LIN {X 0,Y 368.884,Z 241.032,A -85,B 0,C 180,E1 -12733.612,E2 -12733.612} C_VEL
LIN {X 0,Y 368.886,Z 241.019,A -85,B 0,C 180,E1 -12736.692,E2 -12736.692} C_VEL
LIN {X 0,Y 368.885,Z 241.034,A -85,B 0,C 180,E1 -12739.645,E2 -12739.645} C_VEL
LIN {X 0,Y 368.898,Z 241.029,A -85,B 0,C 180,E1 -12743.141,E2 -12743.141} C_VEL
LIN {X 0,Y 368.895,Z 241.032,A -85,B 0,C 180,E1 -12746.458,E2 -12746.458} C_VEL
LIN {X 0,Y 368.911,Z 241.032,A -85,B 0,C 180,E1 -12749.041,E2 -12749.041} C_VEL
LIN {X 0,Y 368.91,Z 241.028,A -85,B 0,C 180,E1 -12751.554,E2 -12751.554} C_VEL
LIN {X 0,Y 368.894,Z 241.03,A -85,B 0,C 180,E1 -12755.216,E2 -12755.216} C_VEL
LIN {X 0,Y 368.894,Z 241.03,A -85,B 0,C 180,E1 -12757.599,E2 -12757.599} C_VEL
LIN {X 0,Y 368.948,Z 241.029,A -85,B 0,C 180,E1 -12761.102,E2 -12761.102} C_VEL
LIN {X 0,Y 368.988,Z 241.017,A -85,B 0,C 180,E1 -12764.531,E2 -12764.531} C_VEL
LIN {X 0,Y 368.993,Z 241.012,A -85,B 0,C 180,E1 -12767.902,E2 -12767.902} C_VEL
LIN {X 0,Y 369.08,Z 241.007,A -85,B 0,C 180,E1 -12771.234,E2 -12771.234} C_VEL
LIN {X 0,Y 369.114,Z 241.004,A -85,B 0,C 180,E1 -12774.533,E2 -12774.533} C_VEL
LIN {X 0,Y 369.281,Z 240.983,A -85,B 0,C 180,E1 -12777.814,E2 -12777.814} C_VEL
LIN {X 0,Y 369.287,Z 240.982,A -85,B 0,C 180,E1 -12782.177,E2 -12782.177} C_VEL
LIN {X 0,Y 369.136,Z 241,A -85,B 0,C 180,E1 -12786.555,E2 -12786.555} C_VEL
LIN {X 0,Y 369.044,Z 241.011,A -85,B 0,C 180,E1 -12789.864,E2 -12789.864} C_VEL
LIN {X 0,Y 369.016,Z 241.014,A -85,B 0,C 180,E1 -12793.768,E2 -12793.768} C_VEL
LIN {X 0,Y 368.968,Z 241.023,A -85,B 0,C 180,E1 -12797.739,E2 -12797.739} C_VEL
LIN {X 0,Y 368.885,Z 241.034,A -85,B 0,C 180,E1 -12801.217,E2 -12801.217} C_VEL
LIN {X 0,Y 368.928,Z 241.026,A -85,B 0,C 180,E1 -12804.772,E2 -12804.772} C_VEL
LIN {X 0,Y 368.935,Z 241.026,A -85,B 0,C 180,E1 -12807.2,E2 -12807.2} C_VEL
LIN {X 0,Y 368.9,Z 241.033,A -85,B 0,C 180,E1 -12810.95,E2 -12810.95} C_VEL
LIN {X 0,Y 368.898,Z 241.029,A -85,B 0,C 180,E1 -12814.998,E2 -12814.998} C_VEL
LIN {X 0,Y 368.88,Z 241.032,A -85,B 0,C 180,E1 -12818.638,E2 -12818.638} C_VEL
LIN {X 0,Y 368.983,Z 241.215,A -85,B 0,C 180,E1 -12821.709,E2 -12821.709} C_VEL
LIN {X 0,Y 371.362,Z 251.966,A -85,B 0,C 180,E1 -12824.763,E2 -12824.763} C_VEL
LIN {X 0,Y 372.623,Z 259.108,A -85,B 0,C 180,E1 -12826.62,E2 -12826.62} C_VEL
LIN {X 0,Y 373.619,Z 263.254,A -85,B 0,C 180,E1 -12826.843,E2 -12826.843} C_VEL
LIN {X 0,Y 377.88,Z 282.484,A -85,B 0,C 180,E1 -12827.564,E2 -12827.564} C_VEL
LIN {X 0,Y 378.656,Z 288.482,A -85,B 0,C 180,E1 -12827.743,E2 -12827.743} C_VEL
LIN {X 0,Y 377.067,Z 367.322,A -85,B 0,C 180,E1 -12829.314,E2 -12829.314} C_VEL
LIN {X 0,Y 376.455,Z 380.341,A -85,B 0,C 180,E1 -12829.785,E2 -12829.785} C_VEL
LIN {X 0,Y 375.568,Z 393.469,A -85,B 0,C 180,E1 -12830.49,E2 -12830.49} C_VEL
LIN {X 0,Y 374.533,Z 405.678,A -85,B 0,C 180,E1 -12831.399,E2 -12831.399} C_VEL
LIN {X 0,Y 373.417,Z 416.7,A -85,B 0,C 180,E1 -12832.453,E2 -12832.453} C_VEL
LIN {X 0,Y 372.202,Z 426.94,A -85,B 0,C 180,E1 -12833.673,E2 -12833.673} C_VEL
LIN {X 0,Y 371.111,Z 436.307,A -85,B 0,C 180,E1 -12835.071,E2 -12835.071} C_VEL
LIN {X 0,Y 370.052,Z 444.979,A -85,B 0,C 180,E1 -12836.672,E2 -12836.672} C_VEL
LIN {X 0,Y 369.106,Z 452.589,A -85,B 0,C 180,E1 -12838.428,E2 -12838.428} C_VEL
LIN {X 0,Y 368.416,Z 458.773,A -85,B 0,C 180,E1 -12840.268,E2 -12840.268} C_VEL
LIN {X 0,Y 367.945,Z 463.489,A -85,B 0,C 180,E1 -12842.1,E2 -12842.1} C_VEL
LIN {X 0,Y 367.538,Z 466.997,A -85,B 0,C 180,E1 -12843.977,E2 -12843.977} C_VEL
LIN {X 0,Y 367.326,Z 468.508,A -85,B 0,C 180,E1 -12845.109,E2 -12845.109} C_VEL
LIN {X 0,Y 367.174,Z 469.903,A -85,B 0,C 180,E1 -12846.729,E2 -12846.729} C_VEL
LIN {X 0,Y 367.102,Z 470.42,A -85,B 0,C 180,E1 -12848.672,E2 -12848.672} C_VEL
LIN {X 0,Y 367.154,Z 470.118,A -85,B 0,C 180,E1 -12849.848,E2 -12849.848} C_VEL
LIN {X 0,Y 367.164,Z 469.396,A -85,B 0,C 180,E1 -12851.012,E2 -12851.012} C_VEL
LIN {X 0,Y 367.341,Z 467.033,A -85,B 0,C 180,E1 -12853.037,E2 -12853.037} C_VEL
LIN {X 0,Y 367.635,Z 463.214,A -85,B 0,C 180,E1 -12855.046,E2 -12855.046} C_VEL
LIN {X 0,Y 367.968,Z 458.316,A -85,B 0,C 180,E1 -12856.896,E2 -12856.896} C_VEL
LIN {X 0,Y 368.487,Z 451.945,A -85,B 0,C 180,E1 -12858.728,E2 -12858.728} C_VEL
LIN {X 0,Y 369.092,Z 444.484,A -85,B 0,C 180,E1 -12860.411,E2 -12860.411} C_VEL
LIN {X 0,Y 369.877,Z 436.445,A -85,B 0,C 180,E1 -12861.876,E2 -12861.876} C_VEL
LIN {X 0,Y 370.717,Z 426.62,A -85,B 0,C 180,E1 -12863.334,E2 -12863.334} C_VEL
LIN {X 0,Y 371.696,Z 416.058,A -85,B 0,C 180,E1 -12864.577,E2 -12864.577} C_VEL
LIN {X 0,Y 372.649,Z 404.329,A -85,B 0,C 180,E1 -12865.675,E2 -12865.675} C_VEL
LIN {X 0,Y 373.338,Z 393.146,A -85,B 0,C 180,E1 -12866.493,E2 -12866.493} C_VEL
LIN {X 0,Y 374.013,Z 380.48,A -85,B 0,C 180,E1 -12867.174,E2 -12867.174} C_VEL
LIN {X 0,Y 374.519,Z 367.44,A -85,B 0,C 180,E1 -12867.649,E2 -12867.649} C_VEL
LIN {X 0,Y 375.577,Z 299.972,A -85,B 0,C 180,E1 -12868.986,E2 -12868.986} C_VEL
LIN {X 0,Y 375.805,Z 285.428,A -85,B 0,C 180,E1 -12869.266,E2 -12869.266} C_VEL
LIN {X 0,Y 371.349,Z 259.539,A -85,B 0,C 180,E1 -12870.036,E2 -12870.036} C_VEL
LIN {X 0,Y 371.475,Z 257.113,A -85,B 0,C 180,E1 -12870.544,E2 -12870.544} C_VEL
LIN {X 0,Y 371.516,Z 253.896,A -85,B 0,C 180,E1 -12871.357,E2 -12871.357} C_VEL
LIN {X 0,Y 369.913,Z 245.755,A -85,B 0,C 180,E1 -12873.542,E2 -12873.542} C_VEL
LIN {X 0,Y 369.638,Z 244.48,A -85,B 0,C 180,E1 -12873.89,E2 -12873.89} C_VEL
LIN {X 0,Y 368.97,Z 242.94,A -85,B 0,C 180,E1 -12874.434,E2 -12874.434} C_VEL
LIN {X 0,Y 367.348,Z 241.756,A -85,B 0,C 180,E1 -12875.294,E2 -12875.294} C_VEL
LIN {X 0,Y 365.439,Z 241.465,A -85,B 0,C 180,E1 -12876.173,E2 -12876.173} C_VEL
LIN {X 0,Y 363.108,Z 241.757,A -85,B 0,C 180,E1 -12877.399,E2 -12877.399} C_VEL
LIN {X 0,Y 362.124,Z 241.878,A -85,B 0,C 180,E1 -12878.345,E2 -12878.345} C_VEL
LIN {X 0,Y 362.031,Z 241.885,A -85,B 0,C 180,E1 -12878.665,E2 -12878.665} C_VEL
LIN {X 0,Y 361.927,Z 241.898,A -85,B 0,C 180,E1 -12882.335,E2 -12882.335} C_VEL
LIN {X 0,Y 361.925,Z 241.898,A -85,B 0,C 180,E1 -12884.624,E2 -12884.624} C_VEL
LIN {X 0,Y 361.92,Z 241.902,A -85,B 0,C 180,E1 -12888.103,E2 -12888.103} C_VEL
LIN {X 0,Y 361.82,Z 241.915,A -85,B 0,C 180,E1 -12891.659,E2 -12891.659} C_VEL
LIN {X 0,Y 361.836,Z 241.909,A -85,B 0,C 180,E1 -12895.299,E2 -12895.299} C_VEL
LIN {X 0,Y 361.825,Z 241.91,A -85,B 0,C 180,E1 -12899.078,E2 -12899.078} C_VEL
LIN {X 0,Y 361.818,Z 241.912,A -85,B 0,C 180,E1 -12902.95,E2 -12902.95} C_VEL
LIN {X 0,Y 361.836,Z 241.909,A -85,B 0,C 180,E1 -12905.642,E2 -12905.642} C_VEL
LIN {X 0,Y 361.799,Z 241.915,A -85,B 0,C 180,E1 -12909.022,E2 -12909.022} C_VEL
LIN {X 0,Y 361.805,Z 241.917,A -85,B 0,C 180,E1 -12912.835,E2 -12912.835} C_VEL
LIN {X 0,Y 361.795,Z 241.914,A -85,B 0,C 180,E1 -12915.952,E2 -12915.952} C_VEL
LIN {X 0,Y 361.794,Z 241.917,A -85,B 0,C 180,E1 -12919.254,E2 -12919.254} C_VEL
LIN {X 0,Y 361.846,Z 241.914,A -85,B 0,C 180,E1 -12922.987,E2 -12922.987} C_VEL
LIN {X 0,Y 361.844,Z 241.91,A -85,B 0,C 180,E1 -12926.637,E2 -12926.637} C_VEL
LIN {X 0,Y 361.836,Z 241.911,A -85,B 0,C 180,E1 -12929.675,E2 -12929.675} C_VEL
LIN {X 0,Y 361.846,Z 241.913,A -85,B 0,C 180,E1 -12933.473,E2 -12933.473} C_VEL
LIN {X 0,Y 361.868,Z 241.909,A -85,B 0,C 180,E1 -12937.149,E2 -12937.149} C_VEL
LIN {X 0,Y 361.88,Z 241.904,A -85,B 0,C 180,E1 -12940.727,E2 -12940.727} C_VEL
LIN {X 0,Y 361.941,Z 241.897,A -85,B 0,C 180,E1 -12944.231,E2 -12944.231} C_VEL
LIN {X 0,Y 361.999,Z 241.889,A -85,B 0,C 180,E1 -12946.533,E2 -12946.533} C_VEL
LIN {X 0,Y 361.997,Z 241.895,A -85,B 0,C 180,E1 -12949.942,E2 -12949.942} C_VEL
LIN {X 0,Y 362.122,Z 241.874,A -85,B 0,C 180,E1 -12953.318,E2 -12953.318} C_VEL
LIN {X 0,Y 362.27,Z 241.858,A -85,B 0,C 180,E1 -12957.781,E2 -12957.781} C_VEL
LIN {X 0,Y 362.207,Z 241.863,A -85,B 0,C 180,E1 -12961.116,E2 -12961.116} C_VEL
LIN {X 0,Y 362.265,Z 241.863,A -85,B 0,C 180,E1 -12962.228,E2 -12962.228} C_VEL
LIN {X 0,Y 362.128,Z 241.876,A -85,B 0,C 180,E1 -12966.691,E2 -12966.691} C_VEL
LIN {X 0,Y 362.008,Z 241.89,A -85,B 0,C 180,E1 -12970.067,E2 -12970.067} C_VEL
LIN {X 0,Y 362.011,Z 241.888,A -85,B 0,C 180,E1 -12973.902,E2 -12973.902} C_VEL
LIN {X 0,Y 361.942,Z 241.9,A -85,B 0,C 180,E1 -12976.937,E2 -12976.937} C_VEL
LIN {X 0,Y 361.901,Z 241.904,A -85,B 0,C 180,E1 -12980.464,E2 -12980.464} C_VEL
LIN {X 0,Y 361.909,Z 241.9,A -85,B 0,C 180,E1 -12984.115,E2 -12984.115} C_VEL
LIN {X 0,Y 361.851,Z 241.908,A -85,B 0,C 180,E1 -12987.787,E2 -12987.787} C_VEL
LIN {X 0,Y 361.864,Z 241.911,A -85,B 0,C 180,E1 -12991.287,E2 -12991.287} C_VEL
LIN {X 0,Y 361.87,Z 241.905,A -85,B 0,C 180,E1 -12994.282,E2 -12994.282} C_VEL
LIN {X 0,Y 361.876,Z 241.909,A -85,B 0,C 180,E1 -12997.223,E2 -12997.223} C_VEL
LIN {X 0,Y 361.827,Z 241.911,A -85,B 0,C 180,E1 -13000.752,E2 -13000.752} C_VEL
LIN {X 0,Y 361.827,Z 241.91,A -85,B 0,C 180,E1 -13004.371,E2 -13004.371} C_VEL
LIN {X 0,Y 361.839,Z 241.914,A -85,B 0,C 180,E1 -13007.572,E2 -13007.572} C_VEL
LIN {X 0,Y 361.86,Z 241.91,A -85,B 0,C 180,E1 -13011.572,E2 -13011.572} C_VEL
LIN {X 0,Y 361.891,Z 241.903,A -85,B 0,C 180,E1 -13014.656,E2 -13014.656} C_VEL
LIN {X 0,Y 361.855,Z 241.912,A -85,B 0,C 180,E1 -13018.371,E2 -13018.371} C_VEL
LIN {X 0,Y 361.932,Z 242.078,A -85,B 0,C 180,E1 -13021.906,E2 -13021.906} C_VEL
LIN {X 0,Y 363.903,Z 251.935,A -85,B 0,C 180,E1 -13024.549,E2 -13024.549} C_VEL
LIN {X 0,Y 364.929,Z 258.159,A -85,B 0,C 180,E1 -13026.143,E2 -13026.143} C_VEL
LIN {X 0,Y 364.18,Z 268.524,A -85,B 0,C 180,E1 -13028.594,E2 -13028.594} C_VEL
LIN {X 0,Y 364.736,Z 272.676,A -85,B 0,C 180,E1 -13028.775,E2 -13028.775} C_VEL
LIN {X 0,Y 368.963,Z 299.983,A -85,B 0,C 180,E1 -13029.539,E2 -13029.539} C_VEL
LIN {X 0,Y 367.671,Z 376.615,A -85,B 0,C 180,E1 -13031.072,E2 -13031.072} C_VEL
LIN {X 0,Y 367.097,Z 389.795,A -85,B 0,C 180,E1 -13031.548,E2 -13031.548} C_VEL
LIN {X 0,Y 366.391,Z 401.948,A -85,B 0,C 180,E1 -13032.198,E2 -13032.198} C_VEL
LIN {X 0,Y 365.439,Z 414.213,A -85,B 0,C 180,E1 -13033.088,E2 -13033.088} C_VEL
LIN {X 0,Y 364.526,Z 425.841,A -85,B 0,C 180,E1 -13034.196,E2 -13034.196} C_VEL
LIN {X 0,Y 363.631,Z 436.307,A -85,B 0,C 180,E1 -13035.447,E2 -13035.447} C_VEL
LIN {X 0,Y 362.755,Z 445.691,A -85,B 0,C 180,E1 -13036.84,E2 -13036.84} C_VEL
LIN {X 0,Y 361.837,Z 454.761,A -85,B 0,C 180,E1 -13038.515,E2 -13038.515} C_VEL
LIN {X 0,Y 361.209,Z 462.062,A -85,B 0,C 180,E1 -13040.196,E2 -13040.196} C_VEL
LIN {X 0,Y 360.825,Z 466.983,A -85,B 0,C 180,E1 -13041.598,E2 -13041.598} C_VEL
LIN {X 0,Y 360.511,Z 471.754,A -85,B 0,C 180,E1 -13043.281,E2 -13043.281} C_VEL
LIN {X 0,Y 360.358,Z 475.394,A -85,B 0,C 180,E1 -13044.963,E2 -13044.963} C_VEL
LIN {X 0,Y 360.28,Z 478.009,A -85,B 0,C 180,E1 -13046.643,E2 -13046.643} C_VEL
LIN {X 0,Y 360.23,Z 479.236,A -85,B 0,C 180,E1 -13047.762,E2 -13047.762} C_VEL
LIN {X 0,Y 360.256,Z 480.037,A -85,B 0,C 180,E1 -13048.88,E2 -13048.88} C_VEL
LIN {X 0,Y 360.281,Z 480.419,A -85,B 0,C 180,E1 -13049.998,E2 -13049.998} C_VEL
LIN {X 0,Y 360.254,Z 480.415,A -85,B 0,C 180,E1 -13051.116,E2 -13051.116} C_VEL
LIN {X 0,Y 360.229,Z 480.027,A -85,B 0,C 180,E1 -13052.234,E2 -13052.234} C_VEL
LIN {X 0,Y 360.283,Z 479.232,A -85,B 0,C 180,E1 -13053.353,E2 -13053.353} C_VEL
LIN {X 0,Y 360.385,Z 478.008,A -85,B 0,C 180,E1 -13054.472,E2 -13054.472} C_VEL
LIN {X 0,Y 360.463,Z 475.575,A -85,B 0,C 180,E1 -13056.072,E2 -13056.072} C_VEL
LIN {X 0,Y 360.789,Z 471.827,A -85,B 0,C 180,E1 -13057.835,E2 -13057.835} C_VEL
LIN {X 0,Y 361.299,Z 467.141,A -85,B 0,C 180,E1 -13059.515,E2 -13059.515} C_VEL
LIN {X 0,Y 362.125,Z 460.107,A -85,B 0,C 180,E1 -13061.472,E2 -13061.472} C_VEL
LIN {X 0,Y 363.127,Z 452.5,A -85,B 0,C 180,E1 -13063.143,E2 -13063.143} C_VEL
LIN {X 0,Y 364.392,Z 443.156,A -85,B 0,C 180,E1 -13064.772,E2 -13064.772} C_VEL
LIN {X 0,Y 365.496,Z 433.562,A -85,B 0,C 180,E1 -13066.13,E2 -13066.13} C_VEL
LIN {X 0,Y 366.714,Z 423.502,A -85,B 0,C 180,E1 -13067.279,E2 -13067.279} C_VEL
LIN {X 0,Y 367.828,Z 413.132,A -85,B 0,C 180,E1 -13068.23,E2 -13068.23} C_VEL
LIN {X 0,Y 368.965,Z 400.702,A -85,B 0,C 180,E1 -13069.108,E2 -13069.108} C_VEL
LIN {X 0,Y 369.847,Z 387.695,A -85,B 0,C 180,E1 -13069.782,E2 -13069.782} C_VEL
LIN {X 0,Y 370.553,Z 374.988,A -85,B 0,C 180,E1 -13070.207,E2 -13070.207} C_VEL
LIN {X 0,Y 371.946,Z 299.95,A -85,B 0,C 180,E1 -13071.731,E2 -13071.731} C_VEL
LIN {X 0,Y 368.448,Z 280.867,A -85,B 0,C 180,E1 -13072.405,E2 -13072.405} C_VEL
LIN {X 0,Y 365.677,Z 268.304,A -85,B 0,C 180,E1 -13072.932,E2 -13072.932} C_VEL
LIN {X 0,Y 366.148,Z 262.196,A -85,B 0,C 180,E1 -13074.371,E2 -13074.371} C_VEL
LIN {X 0,Y 364.501,Z 253.179,A -85,B 0,C 180,E1 -13076.829,E2 -13076.829} C_VEL
LIN {X 0,Y 361.897,Z 242.036,A -85,B 0,C 180,E1 -13080.093,E2 -13080.093} C_VEL
LIN {X 0,Y 361.859,Z 241.909,A -85,B 0,C 180,E1 -13084.277,E2 -13084.277} C_VEL
LIN {X 0,Y 361.864,Z 241.909,A -85,B 0,C 180,E1 -13087.219,E2 -13087.219} C_VEL
LIN {X 0,Y 361.833,Z 241.91,A -85,B 0,C 180,E1 -13090.751,E2 -13090.751} C_VEL
LIN {X 0,Y 361.818,Z 241.917,A -85,B 0,C 180,E1 -13094.365,E2 -13094.365} C_VEL
LIN {X 0,Y 361.831,Z 241.902,A -85,B 0,C 180,E1 -13097.566,E2 -13097.566} C_VEL
LIN {X 0,Y 361.843,Z 241.909,A -85,B 0,C 180,E1 -13101.568,E2 -13101.568} C_VEL
LIN {X 0,Y 361.873,Z 241.907,A -85,B 0,C 180,E1 -13104.652,E2 -13104.652} C_VEL
LIN {X 0,Y 361.836,Z 241.911,A -85,B 0,C 180,E1 -13108.367,E2 -13108.367} C_VEL
LIN {X 0,Y 361.863,Z 241.905,A -85,B 0,C 180,E1 -13110.948,E2 -13110.948} C_VEL
LIN {X 0,Y 361.863,Z 241.904,A -85,B 0,C 180,E1 -13114.701,E2 -13114.701} C_VEL
LIN {X 0,Y 361.849,Z 241.907,A -85,B 0,C 180,E1 -13118.341,E2 -13118.341} C_VEL
LIN {X 0,Y 361.914,Z 241.899,A -85,B 0,C 180,E1 -13122.081,E2 -13122.081} C_VEL
LIN {X 0,Y 361.954,Z 241.9,A -85,B 0,C 180,E1 -13125.375,E2 -13125.375} C_VEL
LIN {X 0,Y 361.958,Z 241.891,A -85,B 0,C 180,E1 -13128.8,E2 -13128.8} C_VEL
LIN {X 0,Y 362.075,Z 241.872,A -85,B 0,C 180,E1 -13132.187,E2 -13132.187} C_VEL
LIN {X 0,Y 362.087,Z 241.879,A -85,B 0,C 180,E1 -13134.427,E2 -13134.427} C_VEL
LIN {X 0,Y 362.243,Z 241.859,A -85,B 0,C 180,E1 -13137.772,E2 -13137.772} C_VEL
LIN {X 0,Y 362.25,Z 241.859,A -85,B 0,C 180,E1 -13142.219,E2 -13142.219} C_VEL
LIN {X 0,Y 362.1,Z 241.876,A -85,B 0,C 180,E1 -13146.683,E2 -13146.683} C_VEL
LIN {X 0,Y 361.98,Z 241.891,A -85,B 0,C 180,E1 -13150.059,E2 -13150.059} C_VEL
LIN {X 0,Y 361.977,Z 241.892,A -85,B 0,C 180,E1 -13153.894,E2 -13153.894} C_VEL
LIN {X 0,Y 361.905,Z 241.899,A -85,B 0,C 180,E1 -13156.93,E2 -13156.93} C_VEL
LIN {X 0,Y 361.862,Z 241.91,A -85,B 0,C 180,E1 -13160.457,E2 -13160.457} C_VEL
LIN {X 0,Y 361.867,Z 241.912,A -85,B 0,C 180,E1 -13164.109,E2 -13164.109} C_VEL
LIN {X 0,Y 361.914,Z 241.903,A -85,B 0,C 180,E1 -13166.717,E2 -13166.717} C_VEL
LIN {X 0,Y 361.843,Z 241.911,A -85,B 0,C 180,E1 -13170.324,E2 -13170.324} C_VEL
LIN {X 0,Y 361.823,Z 241.917,A -85,B 0,C 180,E1 -13174.277,E2 -13174.277} C_VEL
LIN {X 0,Y 361.84,Z 241.914,A -85,B 0,C 180,E1 -13177.221,E2 -13177.221} C_VEL
LIN {X 0,Y 361.925,Z 242.054,A -85,B 0,C 180,E1 -13181.221,E2 -13181.221} C_VEL
LIN {X 0,Y 364.082,Z 251.548,A -85,B 0,C 180,E1 -13184.013,E2 -13184.013} C_VEL
LIN {X 0,Y 365.584,Z 259.305,A -85,B 0,C 180,E1 -13186.095,E2 -13186.095} C_VEL
LIN {X 0,Y 367.171,Z 264.374,A -85,B 0,C 180,E1 -13186.373,E2 -13186.373} C_VEL
LIN {X 0,Y 371.549,Z 284.065,A -85,B 0,C 180,E1 -13187.135,E2 -13187.135} C_VEL
LIN {X 0,Y 372.244,Z 288.032,A -85,B 0,C 180,E1 -13187.272,E2 -13187.272} C_VEL
LIN {X 0,Y 370.567,Z 367.095,A -85,B 0,C 180,E1 -13188.876,E2 -13188.876} C_VEL
LIN {X 0,Y 369.964,Z 379.833,A -85,B 0,C 180,E1 -13189.339,E2 -13189.339} C_VEL
LIN {X 0,Y 369.075,Z 392.402,A -85,B 0,C 180,E1 -13190.011,E2 -13190.011} C_VEL
LIN {X 0,Y 368.166,Z 403.08,A -85,B 0,C 180,E1 -13190.78,E2 -13190.78} C_VEL
LIN {X 0,Y 366.943,Z 414.608,A -85,B 0,C 180,E1 -13191.844,E2 -13191.844} C_VEL
LIN {X 0,Y 365.696,Z 425.274,A -85,B 0,C 180,E1 -13193.092,E2 -13193.092} C_VEL
LIN {X 0,Y 364.511,Z 434.505,A -85,B 0,C 180,E1 -13194.427,E2 -13194.427} C_VEL
LIN {X 0,Y 363.477,Z 442.768,A -85,B 0,C 180,E1 -13195.896,E2 -13195.896} C_VEL
LIN {X 0,Y 362.533,Z 449.914,A -85,B 0,C 180,E1 -13197.458,E2 -13197.458} C_VEL
LIN {X 0,Y 361.725,Z 456.172,A -85,B 0,C 180,E1 -13199.158,E2 -13199.158} C_VEL
LIN {X 0,Y 361.097,Z 461.808,A -85,B 0,C 180,E1 -13201.13,E2 -13201.13} C_VEL
LIN {X 0,Y 360.696,Z 465.301,A -85,B 0,C 180,E1 -13202.751,E2 -13202.751} C_VEL
LIN {X 0,Y 360.309,Z 468.147,A -85,B 0,C 180,E1 -13204.59,E2 -13204.59} C_VEL
LIN {X 0,Y 360.078,Z 469.937,A -85,B 0,C 180,E1 -13206.525,E2 -13206.525} C_VEL
LIN {X 0,Y 360.017,Z 470.506,A -85,B 0,C 180,E1 -13208.231,E2 -13208.231} C_VEL
LIN {X 0,Y 360.047,Z 470.337,A -85,B 0,C 180,E1 -13209.526,E2 -13209.526} C_VEL
LIN {X 0,Y 360.049,Z 469.76,A -85,B 0,C 180,E1 -13210.622,E2 -13210.622} C_VEL
LIN {X 0,Y 360.09,Z 468.721,A -85,B 0,C 180,E1 -13211.805,E2 -13211.805} C_VEL
LIN {X 0,Y 360.231,Z 467.239,A -85,B 0,C 180,E1 -13212.986,E2 -13212.986} C_VEL
LIN {X 0,Y 360.477,Z 464.114,A -85,B 0,C 180,E1 -13214.742,E2 -13214.742} C_VEL
LIN {X 0,Y 360.873,Z 458.918,A -85,B 0,C 180,E1 -13216.814,E2 -13216.814} C_VEL
LIN {X 0,Y 361.406,Z 452.311,A -85,B 0,C 180,E1 -13218.789,E2 -13218.789} C_VEL
LIN {X 0,Y 362.029,Z 444.907,A -85,B 0,C 180,E1 -13220.504,E2 -13220.504} C_VEL
LIN {X 0,Y 362.939,Z 435.68,A -85,B 0,C 180,E1 -13222.211,E2 -13222.211} C_VEL
LIN {X 0,Y 363.795,Z 426.139,A -85,B 0,C 180,E1 -13223.624,E2 -13223.624} C_VEL
LIN {X 0,Y 364.839,Z 415.442,A -85,B 0,C 180,E1 -13224.89,E2 -13224.89} C_VEL
LIN {X 0,Y 365.827,Z 403.481,A -85,B 0,C 180,E1 -13226.014,E2 -13226.014} C_VEL
LIN {X 0,Y 366.604,Z 390.865,A -85,B 0,C 180,E1 -13226.911,E2 -13226.911} C_VEL
LIN {X 0,Y 367.296,Z 378.133,A -85,B 0,C 180,E1 -13227.569,E2 -13227.569} C_VEL
LIN {X 0,Y 367.743,Z 364.816,A -85,B 0,C 180,E1 -13228.017,E2 -13228.017} C_VEL
LIN {X 0,Y 369.04,Z 286.728,A -85,B 0,C 180,E1 -13229.566,E2 -13229.566} C_VEL
LIN {X 0,Y 364.472,Z 259.735,A -85,B 0,C 180,E1 -13230.382,E2 -13230.382} C_VEL
LIN {X 0,Y 364.479,Z 258.385,A -85,B 0,C 180,E1 -13230.609,E2 -13230.609} C_VEL
LIN {X 0,Y 364.573,Z 255.361,A -85,B 0,C 180,E1 -13231.382,E2 -13231.382} C_VEL
LIN {X 0,Y 362.982,Z 247.218,A -85,B 0,C 180,E1 -13233.609,E2 -13233.609} C_VEL
LIN {X 0,Y 362.022,Z 241.921,A -85,B 0,C 180,E1 -13235.153,E2 -13235.153} C_VEL
LIN {X 0,Y 362.076,Z 241.88,A -85,B 0,C 180,E1 -13238.186,E2 -13238.186} C_VEL
LIN {X 0,Y 362.031,Z 241.885,A -85,B 0,C 180,E1 -13238.665,E2 -13238.665} C_VEL
LIN {X 0,Y 361.311,Z 241.981,A -85,B 0,C 180,E1 -13239.593,E2 -13239.593} C_VEL
LIN {X 0,Y 358.39,Z 242.34,A -85,B 0,C 180,E1 -13241.1,E2 -13241.1} C_VEL
LIN {X 0,Y 355.965,Z 242.641,A -85,B 0,C 180,E1 -13242.32,E2 -13242.32} C_VEL
LIN {X 0,Y 354.964,Z 242.768,A -85,B 0,C 180,E1 -13243.265,E2 -13243.265} C_VEL
LIN {X 0,Y 354.902,Z 242.777,A -85,B 0,C 180,E1 -13243.584,E2 -13243.584} C_VEL
LIN {X 0,Y 354.862,Z 242.779,A -85,B 0,C 180,E1 -13247.284,E2 -13247.284} C_VEL
LIN {X 0,Y 354.791,Z 242.787,A -85,B 0,C 180,E1 -13250.891,E2 -13250.891} C_VEL
LIN {X 0,Y 354.78,Z 242.789,A -85,B 0,C 180,E1 -13254.584,E2 -13254.584} C_VEL
LIN {X 0,Y 354.77,Z 242.793,A -85,B 0,C 180,E1 -13258.39,E2 -13258.39} C_VEL
LIN {X 0,Y 354.755,Z 242.797,A -85,B 0,C 180,E1 -13262.338,E2 -13262.338} C_VEL
LIN {X 0,Y 354.79,Z 242.787,A -85,B 0,C 180,E1 -13265.703,E2 -13265.703} C_VEL
LIN {X 0,Y 354.744,Z 242.792,A -85,B 0,C 180,E1 -13269.417,E2 -13269.417} C_VEL
LIN {X 0,Y 354.758,Z 242.795,A -85,B 0,C 180,E1 -13272.871,E2 -13272.871} C_VEL
LIN {X 0,Y 354.744,Z 242.793,A -85,B 0,C 180,E1 -13276.108,E2 -13276.108} C_VEL
LIN {X 0,Y 354.747,Z 242.795,A -85,B 0,C 180,E1 -13279.181,E2 -13279.181} C_VEL
LIN {X 0,Y 354.783,Z 242.789,A -85,B 0,C 180,E1 -13282.41,E2 -13282.41} C_VEL
LIN {X 0,Y 354.794,Z 242.792,A -85,B 0,C 180,E1 -13284.946,E2 -13284.946} C_VEL
LIN {X 0,Y 354.778,Z 242.789,A -85,B 0,C 180,E1 -13288.412,E2 -13288.412} C_VEL
LIN {X 0,Y 354.779,Z 242.791,A -85,B 0,C 180,E1 -13291.619,E2 -13291.619} C_VEL
LIN {X 0,Y 354.797,Z 242.792,A -85,B 0,C 180,E1 -13295.425,E2 -13295.425} C_VEL
LIN {X 0,Y 354.821,Z 242.786,A -85,B 0,C 180,E1 -13299.118,E2 -13299.118} C_VEL
LIN {X 0,Y 354.878,Z 242.776,A -85,B 0,C 180,E1 -13302.724,E2 -13302.724} C_VEL
LIN {X 0,Y 354.951,Z 242.768,A -85,B 0,C 180,E1 -13306.26,E2 -13306.26} C_VEL
LIN {X 0,Y 354.953,Z 242.772,A -85,B 0,C 180,E1 -13309.74,E2 -13309.74} C_VEL
LIN {X 0,Y 355.088,Z 242.75,A -85,B 0,C 180,E1 -13313.185,E2 -13313.185} C_VEL
LIN {X 0,Y 355.232,Z 242.735,A -85,B 0,C 180,E1 -13317.737,E2 -13317.737} C_VEL
LIN {X 0,Y 355.176,Z 242.739,A -85,B 0,C 180,E1 -13321.138,E2 -13321.138} C_VEL
LIN {X 0,Y 355.227,Z 242.739,A -85,B 0,C 180,E1 -13322.272,E2 -13322.272} C_VEL
LIN {X 0,Y 355.095,Z 242.751,A -85,B 0,C 180,E1 -13326.824,E2 -13326.824} C_VEL
LIN {X 0,Y 354.965,Z 242.769,A -85,B 0,C 180,E1 -13330.269,E2 -13330.269} C_VEL
LIN {X 0,Y 354.956,Z 242.767,A -85,B 0,C 180,E1 -13334.022,E2 -13334.022} C_VEL
LIN {X 0,Y 354.904,Z 242.773,A -85,B 0,C 180,E1 -13338.095,E2 -13338.095} C_VEL
LIN {X 0,Y 354.829,Z 242.782,A -85,B 0,C 180,E1 -13342.11,E2 -13342.11} C_VEL
LIN {X 0,Y 354.864,Z 242.78,A -85,B 0,C 180,E1 -13344.58,E2 -13344.58} C_VEL
LIN {X 0,Y 354.813,Z 242.784,A -85,B 0,C 180,E1 -13348.388,E2 -13348.388} C_VEL
LIN {X 0,Y 354.803,Z 242.785,A -85,B 0,C 180,E1 -13352.336,E2 -13352.336} C_VEL
LIN {X 0,Y 354.838,Z 242.783,A -85,B 0,C 180,E1 -13355.701,E2 -13355.701} C_VEL
LIN {X 0,Y 354.786,Z 242.794,A -85,B 0,C 180,E1 -13359.414,E2 -13359.414} C_VEL
LIN {X 0,Y 354.798,Z 242.786,A -85,B 0,C 180,E1 -13362.867,E2 -13362.867} C_VEL
LIN {X 0,Y 354.778,Z 242.79,A -85,B 0,C 180,E1 -13366.103,E2 -13366.103} C_VEL
LIN {X 0,Y 354.779,Z 242.789,A -85,B 0,C 180,E1 -13369.176,E2 -13369.176} C_VEL
LIN {X 0,Y 354.817,Z 242.785,A -85,B 0,C 180,E1 -13372.405,E2 -13372.405} C_VEL
LIN {X 0,Y 354.829,Z 242.782,A -85,B 0,C 180,E1 -13374.941,E2 -13374.941} C_VEL
LIN {X 0,Y 354.81,Z 242.789,A -85,B 0,C 180,E1 -13378.405,E2 -13378.405} C_VEL
LIN {X 0,Y 354.889,Z 242.923,A -85,B 0,C 180,E1 -13381.621,E2 -13381.621} C_VEL
LIN {X 0,Y 356.836,Z 252.758,A -85,B 0,C 180,E1 -13384.321,E2 -13384.321} C_VEL
LIN {X 0,Y 357.922,Z 258.976,A -85,B 0,C 180,E1 -13385.954,E2 -13385.954} C_VEL
LIN {X 0,Y 357.45,Z 265.998,A -85,B 0,C 180,E1 -13387.68,E2 -13387.68} C_VEL
LIN {X 0,Y 357.318,Z 268.816,A -85,B 0,C 180,E1 -13388.274,E2 -13388.274} C_VEL
LIN {X 0,Y 359.225,Z 281.426,A -85,B 0,C 180,E1 -13388.678,E2 -13388.678} C_VEL
LIN {X 0,Y 362.172,Z 300.669,A -85,B 0,C 180,E1 -13389.226,E2 -13389.226} C_VEL
LIN {X 0,Y 360.856,Z 376.741,A -85,B 0,C 180,E1 -13390.774,E2 -13390.774} C_VEL
LIN {X 0,Y 360.26,Z 389.844,A -85,B 0,C 180,E1 -13391.258,E2 -13391.258} C_VEL
LIN {X 0,Y 359.529,Z 401.958,A -85,B 0,C 180,E1 -13391.92,E2 -13391.92} C_VEL
LIN {X 0,Y 358.639,Z 413.39,A -85,B 0,C 180,E1 -13392.757,E2 -13392.757} C_VEL
LIN {X 0,Y 357.648,Z 425.153,A -85,B 0,C 180,E1 -13393.883,E2 -13393.883} C_VEL
LIN {X 0,Y 356.726,Z 435.722,A -85,B 0,C 180,E1 -13395.158,E2 -13395.158} C_VEL
LIN {X 0,Y 355.794,Z 445.22,A -85,B 0,C 180,E1 -13396.578,E2 -13396.578} C_VEL
LIN {X 0,Y 354.843,Z 454.355,A -85,B 0,C 180,E1 -13398.285,E2 -13398.285} C_VEL
LIN {X 0,Y 354.186,Z 461.711,A -85,B 0,C 180,E1 -13400,E2 -13400} C_VEL
LIN {X 0,Y 353.762,Z 466.679,A -85,B 0,C 180,E1 -13401.429,E2 -13401.429} C_VEL
LIN {X 0,Y 353.43,Z 471.495,A -85,B 0,C 180,E1 -13403.146,E2 -13403.146} C_VEL
LIN {X 0,Y 353.263,Z 475.176,A -85,B 0,C 180,E1 -13404.862,E2 -13404.862} C_VEL
LIN {X 0,Y 353.204,Z 477.829,A -85,B 0,C 180,E1 -13406.576,E2 -13406.576} C_VEL
LIN {X 0,Y 353.141,Z 479.075,A -85,B 0,C 180,E1 -13407.717,E2 -13407.717} C_VEL
LIN {X 0,Y 353.155,Z 479.911,A -85,B 0,C 180,E1 -13408.858,E2 -13408.858} C_VEL
LIN {X 0,Y 353.182,Z 480.311,A -85,B 0,C 180,E1 -13409.998,E2 -13409.998} C_VEL
LIN {X 0,Y 353.154,Z 480.325,A -85,B 0,C 180,E1 -13411.139,E2 -13411.139} C_VEL
LIN {X 0,Y 353.208,Z 479.191,A -85,B 0,C 180,E1 -13413.42,E2 -13413.42} C_VEL
LIN {X 0,Y 353.3,Z 477.988,A -85,B 0,C 180,E1 -13414.562,E2 -13414.562} C_VEL
LIN {X 0,Y 353.363,Z 475.886,A -85,B 0,C 180,E1 -13416.021,E2 -13416.021} C_VEL
LIN {X 0,Y 353.74,Z 471.882,A -85,B 0,C 180,E1 -13417.992,E2 -13417.992} C_VEL
LIN {X 0,Y 354.281,Z 467.237,A -85,B 0,C 180,E1 -13419.706,E2 -13419.706} C_VEL
LIN {X 0,Y 355.149,Z 460.247,A -85,B 0,C 180,E1 -13421.701,E2 -13421.701} C_VEL
LIN {X 0,Y 356.228,Z 452.696,A -85,B 0,C 180,E1 -13423.402,E2 -13423.402} C_VEL
LIN {X 0,Y 357.519,Z 443.588,A -85,B 0,C 180,E1 -13425.041,E2 -13425.041} C_VEL
LIN {X 0,Y 358.701,Z 433.965,A -85,B 0,C 180,E1 -13426.444,E2 -13426.444} C_VEL
LIN {X 0,Y 359.979,Z 424.032,A -85,B 0,C 180,E1 -13427.613,E2 -13427.613} C_VEL
LIN {X 0,Y 361.138,Z 413.843,A -85,B 0,C 180,E1 -13428.58,E2 -13428.58} C_VEL
LIN {X 0,Y 362.325,Z 401.763,A -85,B 0,C 180,E1 -13429.472,E2 -13429.472} C_VEL
LIN {X 0,Y 363.221,Z 389.161,A -85,B 0,C 180,E1 -13430.159,E2 -13430.159} C_VEL
LIN {X 0,Y 364.037,Z 376.07,A -85,B 0,C 180,E1 -13430.628,E2 -13430.628} C_VEL
LIN {X 0,Y 365.518,Z 300.705,A -85,B 0,C 180,E1 -13432.194,E2 -13432.194} C_VEL
LIN {X 0,Y 361.522,Z 279.337,A -85,B 0,C 180,E1 -13432.978,E2 -13432.978} C_VEL
LIN {X 0,Y 358.999,Z 268.251,A -85,B 0,C 180,E1 -13433.467,E2 -13433.467} C_VEL
LIN {X 0,Y 359.27,Z 263.646,A -85,B 0,C 180,E1 -13434.561,E2 -13434.561} C_VEL
LIN {X 0,Y 357.309,Z 253.342,A -85,B 0,C 180,E1 -13437.445,E2 -13437.445} C_VEL
LIN {X 0,Y 354.879,Z 243.126,A -85,B 0,C 180,E1 -13440.493,E2 -13440.493} C_VEL
LIN {X 0,Y 354.805,Z 242.787,A -85,B 0,C 180,E1 -13440.996,E2 -13440.996} C_VEL
LIN {X 0,Y 354.812,Z 242.789,A -85,B 0,C 180,E1 -13443.699,E2 -13443.699} C_VEL
LIN {X 0,Y 354.801,Z 242.792,A -85,B 0,C 180,E1 -13446.457,E2 -13446.457} C_VEL
LIN {X 0,Y 354.803,Z 242.786,A -85,B 0,C 180,E1 -13449.415,E2 -13449.415} C_VEL
LIN {X 0,Y 354.788,Z 242.783,A -85,B 0,C 180,E1 -13452.863,E2 -13452.863} C_VEL
LIN {X 0,Y 354.767,Z 242.779,A -85,B 0,C 180,E1 -13456.1,E2 -13456.1} C_VEL
LIN {X 0,Y 354.767,Z 242.793,A -85,B 0,C 180,E1 -13459.172,E2 -13459.172} C_VEL
LIN {X 0,Y 354.8,Z 242.792,A -85,B 0,C 180,E1 -13462.401,E2 -13462.401} C_VEL
LIN {X 0,Y 354.811,Z 242.789,A -85,B 0,C 180,E1 -13464.937,E2 -13464.937} C_VEL
LIN {X 0,Y 354.792,Z 242.789,A -85,B 0,C 180,E1 -13468.401,E2 -13468.401} C_VEL
LIN {X 0,Y 354.797,Z 242.786,A -85,B 0,C 180,E1 -13471.611,E2 -13471.611} C_VEL
LIN {X 0,Y 354.802,Z 242.786,A -85,B 0,C 180,E1 -13475.416,E2 -13475.416} C_VEL
LIN {X 0,Y 354.82,Z 242.78,A -85,B 0,C 180,E1 -13479.109,E2 -13479.109} C_VEL
LIN {X 0,Y 354.873,Z 242.775,A -85,B 0,C 180,E1 -13482.715,E2 -13482.715} C_VEL
LIN {X 0,Y 354.943,Z 242.769,A -85,B 0,C 180,E1 -13486.251,E2 -13486.251} C_VEL
LIN {X 0,Y 354.944,Z 242.771,A -85,B 0,C 180,E1 -13489.731,E2 -13489.731} C_VEL
LIN {X 0,Y 355.092,Z 242.745,A -85,B 0,C 180,E1 -13493.176,E2 -13493.176} C_VEL
LIN {X 0,Y 355.205,Z 242.734,A -85,B 0,C 180,E1 -13497.728,E2 -13497.728} C_VEL
LIN {X 0,Y 355.129,Z 242.741,A -85,B 0,C 180,E1 -13501.13,E2 -13501.13} C_VEL
LIN {X 0,Y 355.212,Z 242.735,A -85,B 0,C 180,E1 -13502.263,E2 -13502.263} C_VEL
LIN {X 0,Y 355.067,Z 242.753,A -85,B 0,C 180,E1 -13506.816,E2 -13506.816} C_VEL
LIN {X 0,Y 354.936,Z 242.77,A -85,B 0,C 180,E1 -13510.26,E2 -13510.26} C_VEL
LIN {X 0,Y 354.922,Z 242.772,A -85,B 0,C 180,E1 -13514.014,E2 -13514.014} C_VEL
LIN {X 0,Y 354.867,Z 242.784,A -85,B 0,C 180,E1 -13518.088,E2 -13518.088} C_VEL
LIN {X 0,Y 354.794,Z 242.79,A -85,B 0,C 180,E1 -13521.414,E2 -13521.414} C_VEL
LIN {X 0,Y 354.834,Z 242.783,A -85,B 0,C 180,E1 -13524.572,E2 -13524.572} C_VEL
LIN {X 0,Y 354.854,Z 242.781,A -85,B 0,C 180,E1 -13527.092,E2 -13527.092} C_VEL
LIN {X 0,Y 354.77,Z 242.793,A -85,B 0,C 180,E1 -13530.995,E2 -13530.995} C_VEL
LIN {X 0,Y 354.776,Z 242.791,A -85,B 0,C 180,E1 -13533.698,E2 -13533.698} C_VEL
LIN {X 0,Y 354.769,Z 242.789,A -85,B 0,C 180,E1 -13536.456,E2 -13536.456} C_VEL
LIN {X 0,Y 354.872,Z 242.915,A -85,B 0,C 180,E1 -13540.708,E2 -13540.708} C_VEL
LIN {X 0,Y 357.04,Z 252.236,A -85,B 0,C 180,E1 -13543.538,E2 -13543.538} C_VEL
LIN {X 0,Y 358.457,Z 259.388,A -85,B 0,C 180,E1 -13545.52,E2 -13545.52} C_VEL
LIN {X 0,Y 360.825,Z 265.835,A -85,B 0,C 180,E1 -13545.9,E2 -13545.9} C_VEL
LIN {X 0,Y 365.19,Z 285.307,A -85,B 0,C 180,E1 -13546.68,E2 -13546.68} C_VEL
LIN {X 0,Y 365.824,Z 290.408,A -85,B 0,C 180,E1 -13546.841,E2 -13546.841} C_VEL
LIN {X 0,Y 364.084,Z 367.421,A -85,B 0,C 180,E1 -13548.432,E2 -13548.432} C_VEL
LIN {X 0,Y 363.413,Z 380.529,A -85,B 0,C 180,E1 -13548.921,E2 -13548.921} C_VEL
LIN {X 0,Y 362.52,Z 392.758,A -85,B 0,C 180,E1 -13549.594,E2 -13549.594} C_VEL
LIN {X 0,Y 361.483,Z 404.193,A -85,B 0,C 180,E1 -13550.443,E2 -13550.443} C_VEL
LIN {X 0,Y 360.196,Z 415.649,A -85,B 0,C 180,E1 -13551.545,E2 -13551.545} C_VEL
LIN {X 0,Y 358.813,Z 426.786,A -85,B 0,C 180,E1 -13552.902,E2 -13552.902} C_VEL
LIN {X 0,Y 357.6,Z 435.51,A -85,B 0,C 180,E1 -13554.222,E2 -13554.222} C_VEL
LIN {X 0,Y 356.38,Z 444.471,A -85,B 0,C 180,E1 -13555.909,E2 -13555.909} C_VEL
LIN {X 0,Y 355.311,Z 452.181,A -85,B 0,C 180,E1 -13557.722,E2 -13557.722} C_VEL
LIN {X 0,Y 354.489,Z 458.527,A -85,B 0,C 180,E1 -13559.634,E2 -13559.634} C_VEL
LIN {X 0,Y 353.917,Z 463.35,A -85,B 0,C 180,E1 -13561.54,E2 -13561.54} C_VEL
LIN {X 0,Y 353.46,Z 466.908,A -85,B 0,C 180,E1 -13563.463,E2 -13563.463} C_VEL
LIN {X 0,Y 353.099,Z 469.165,A -85,B 0,C 180,E1 -13565.295,E2 -13565.295} C_VEL
LIN {X 0,Y 353.004,Z 470.119,A -85,B 0,C 180,E1 -13566.538,E2 -13566.538} C_VEL
LIN {X 0,Y 352.916,Z 470.555,A -85,B 0,C 180,E1 -13567.77,E2 -13567.77} C_VEL
LIN {X 0,Y 352.938,Z 470.484,A -85,B 0,C 180,E1 -13569.356,E2 -13569.356} C_VEL
LIN {X 0,Y 352.962,Z 469.19,A -85,B 0,C 180,E1 -13571.425,E2 -13571.425} C_VEL
LIN {X 0,Y 353.114,Z 467.624,A -85,B 0,C 180,E1 -13572.79,E2 -13572.79} C_VEL
LIN {X 0,Y 353.352,Z 464.921,A -85,B 0,C 180,E1 -13574.426,E2 -13574.426} C_VEL
LIN {X 0,Y 353.657,Z 460.927,A -85,B 0,C 180,E1 -13576.206,E2 -13576.206} C_VEL
LIN {X 0,Y 354.051,Z 455.748,A -85,B 0,C 180,E1 -13577.972,E2 -13577.972} C_VEL
LIN {X 0,Y 354.622,Z 449.207,A -85,B 0,C 180,E1 -13579.727,E2 -13579.727} C_VEL
LIN {X 0,Y 355.45,Z 440.545,A -85,B 0,C 180,E1 -13581.559,E2 -13581.559} C_VEL
LIN {X 0,Y 356.281,Z 432.596,A -85,B 0,C 180,E1 -13582.92,E2 -13582.92} C_VEL
LIN {X 0,Y 357.248,Z 422.332,A -85,B 0,C 180,E1 -13584.357,E2 -13584.357} C_VEL
LIN {X 0,Y 358.363,Z 410.613,A -85,B 0,C 180,E1 -13585.644,E2 -13585.644} C_VEL
LIN {X 0,Y 359.262,Z 399.116,A -85,B 0,C 180,E1 -13586.637,E2 -13586.637} C_VEL
LIN {X 0,Y 360.003,Z 387.314,A -85,B 0,C 180,E1 -13587.414,E2 -13587.414} C_VEL
LIN {X 0,Y 360.626,Z 373.71,A -85,B 0,C 180,E1 -13588.047,E2 -13588.047} C_VEL
LIN {X 0,Y 360.988,Z 361.728,A -85,B 0,C 180,E1 -13588.398,E2 -13588.398} C_VEL
LIN {X 0,Y 362.234,Z 287.197,A -85,B 0,C 180,E1 -13589.896,E2 -13589.896} C_VEL
LIN {X 0,Y 357.562,Z 259.656,A -85,B 0,C 180,E1 -13590.748,E2 -13590.748} C_VEL
LIN {X 0,Y 357.625,Z 256.818,A -85,B 0,C 180,E1 -13591.409,E2 -13591.409} C_VEL
LIN {X 0,Y 356.044,Z 248.612,A -85,B 0,C 180,E1 -13593.68,E2 -13593.68} C_VEL
LIN {X 0,Y 355.045,Z 243.078,A -85,B 0,C 180,E1 -13595.255,E2 -13595.255} C_VEL
LIN {X 0,Y 355.049,Z 242.758,A -85,B 0,C 180,E1 -13595.682,E2 -13595.682} C_VEL
LIN {X 0,Y 354.992,Z 242.762,A -85,B 0,C 180,E1 -13598.65,E2 -13598.65} C_VEL
LIN {X 0,Y 354.887,Z 242.775,A -85,B 0,C 180,E1 -13602.584,E2 -13602.584} C_VEL
LIN {X 0,Y 354.902,Z 242.777,A -85,B 0,C 180,E1 -13603.584,E2 -13603.584} C_VEL
LIN {X 0,Y 354.291,Z 242.86,A -85,B 0,C 180,E1 -13604.531,E2 -13604.531} C_VEL
LIN {X 0,Y 351.463,Z 243.213,A -85,B 0,C 180,E1 -13606.07,E2 -13606.07} C_VEL
LIN {X 0,Y 349.014,Z 243.513,A -85,B 0,C 180,E1 -13607.315,E2 -13607.315} C_VEL
LIN {X 0,Y 347.932,Z 243.644,A -85,B 0,C 180,E1 -13608.279,E2 -13608.279} C_VEL
LIN {X 0,Y 347.829,Z 243.654,A -85,B 0,C 180,E1 -13608.606,E2 -13608.606} C_VEL
LIN {X 0,Y 347.716,Z 243.669,A -85,B 0,C 180,E1 -13612.585,E2 -13612.585} C_VEL
LIN {X 0,Y 347.713,Z 243.668,A -85,B 0,C 180,E1 -13615.118,E2 -13615.118} C_VEL
LIN {X 0,Y 347.706,Z 243.671,A -85,B 0,C 180,E1 -13617.705,E2 -13617.705} C_VEL
LIN {X 0,Y 347.705,Z 243.674,A -85,B 0,C 180,E1 -13620.354,E2 -13620.354} C_VEL
LIN {X 0,Y 347.72,Z 243.671,A -85,B 0,C 180,E1 -13624.048,E2 -13624.048} C_VEL
LIN {X 0,Y 347.728,Z 243.666,A -85,B 0,C 180,E1 -13627.327,E2 -13627.327} C_VEL
LIN {X 0,Y 347.671,Z 243.677,A -85,B 0,C 180,E1 -13630.307,E2 -13630.307} C_VEL
LIN {X 0,Y 347.698,Z 243.67,A -85,B 0,C 180,E1 -13633.414,E2 -13633.414} C_VEL
LIN {X 0,Y 347.704,Z 243.676,A -85,B 0,C 180,E1 -13636.692,E2 -13636.692} C_VEL
LIN {X 0,Y 347.684,Z 243.672,A -85,B 0,C 180,E1 -13640.188,E2 -13640.188} C_VEL
LIN {X 0,Y 347.739,Z 243.669,A -85,B 0,C 180,E1 -13642.684,E2 -13642.684} C_VEL
LIN {X 0,Y 347.735,Z 243.666,A -85,B 0,C 180,E1 -13645.962,E2 -13645.962} C_VEL
LIN {X 0,Y 347.724,Z 243.668,A -85,B 0,C 180,E1 -13649.656,E2 -13649.656} C_VEL
LIN {X 0,Y 347.726,Z 243.67,A -85,B 0,C 180,E1 -13653.605,E2 -13653.605} C_VEL
LIN {X 0,Y 347.745,Z 243.665,A -85,B 0,C 180,E1 -13656.165,E2 -13656.165} C_VEL
LIN {X 0,Y 347.782,Z 243.662,A -85,B 0,C 180,E1 -13659.913,E2 -13659.913} C_VEL
LIN {X 0,Y 347.83,Z 243.659,A -85,B 0,C 180,E1 -13663.574,E2 -13663.574} C_VEL
LIN {X 0,Y 347.888,Z 243.647,A -85,B 0,C 180,E1 -13667.166,E2 -13667.166} C_VEL
LIN {X 0,Y 347.936,Z 243.641,A -85,B 0,C 180,E1 -13670.706,E2 -13670.706} C_VEL
LIN {X 0,Y 348.04,Z 243.631,A -85,B 0,C 180,E1 -13674.21,E2 -13674.21} C_VEL
LIN {X 0,Y 348.194,Z 243.61,A -85,B 0,C 180,E1 -13677.691,E2 -13677.691} C_VEL
LIN {X 0,Y 348.145,Z 243.614,A -85,B 0,C 180,E1 -13681.161,E2 -13681.161} C_VEL
LIN {X 0,Y 348.188,Z 243.615,A -85,B 0,C 180,E1 -13682.318,E2 -13682.318} C_VEL
LIN {X 0,Y 348.062,Z 243.626,A -85,B 0,C 180,E1 -13686.963,E2 -13686.963} C_VEL
LIN {X 0,Y 347.905,Z 243.65,A -85,B 0,C 180,E1 -13690.479,E2 -13690.479} C_VEL
LIN {X 0,Y 347.913,Z 243.645,A -85,B 0,C 180,E1 -13694.153,E2 -13694.153} C_VEL
LIN {X 0,Y 347.844,Z 243.654,A -85,B 0,C 180,E1 -13698.262,E2 -13698.262} C_VEL
LIN {X 0,Y 347.782,Z 243.66,A -85,B 0,C 180,E1 -13701.629,E2 -13701.629} C_VEL
LIN {X 0,Y 347.782,Z 243.665,A -85,B 0,C 180,E1 -13705.115,E2 -13705.115} C_VEL
LIN {X 0,Y 347.761,Z 243.668,A -85,B 0,C 180,E1 -13709.018,E2 -13709.018} C_VEL
LIN {X 0,Y 347.755,Z 243.664,A -85,B 0,C 180,E1 -13711.916,E2 -13711.916} C_VEL
LIN {X 0,Y 347.804,Z 243.658,A -85,B 0,C 180,E1 -13715.877,E2 -13715.877} C_VEL
LIN {X 0,Y 347.748,Z 243.665,A -85,B 0,C 180,E1 -13718.797,E2 -13718.797} C_VEL
LIN {X 0,Y 347.757,Z 243.666,A -85,B 0,C 180,E1 -13721.833,E2 -13721.833} C_VEL
LIN {X 0,Y 347.716,Z 243.669,A -85,B 0,C 180,E1 -13725.029,E2 -13725.029} C_VEL
LIN {X 0,Y 347.755,Z 243.664,A -85,B 0,C 180,E1 -13728.401,E2 -13728.401} C_VEL
LIN {X 0,Y 347.78,Z 243.665,A -85,B 0,C 180,E1 -13732.014,E2 -13732.014} C_VEL
LIN {X 0,Y 347.762,Z 243.664,A -85,B 0,C 180,E1 -13735.536,E2 -13735.536} C_VEL
LIN {X 0,Y 347.762,Z 243.667,A -85,B 0,C 180,E1 -13738.3,E2 -13738.3} C_VEL
LIN {X 0,Y 347.823,Z 243.756,A -85,B 0,C 180,E1 -13741.32,E2 -13741.32} C_VEL
LIN {X 0,Y 349.909,Z 254.219,A -85,B 0,C 180,E1 -13744.262,E2 -13744.262} C_VEL
LIN {X 0,Y 350.991,Z 261.027,A -85,B 0,C 180,E1 -13746.078,E2 -13746.078} C_VEL
LIN {X 0,Y 350.388,Z 268.562,A -85,B 0,C 180,E1 -13747.888,E2 -13747.888} C_VEL
LIN {X 0,Y 351.568,Z 276.386,A -85,B 0,C 180,E1 -13748.169,E2 -13748.169} C_VEL
LIN {X 0,Y 355.409,Z 301.551,A -85,B 0,C 180,E1 -13748.907,E2 -13748.907} C_VEL
LIN {X 0,Y 354.045,Z 376.864,A -85,B 0,C 180,E1 -13750.465,E2 -13750.465} C_VEL
LIN {X 0,Y 353.436,Z 389.894,A -85,B 0,C 180,E1 -13750.958,E2 -13750.958} C_VEL
LIN {X 0,Y 352.67,Z 401.968,A -85,B 0,C 180,E1 -13751.631,E2 -13751.631} C_VEL
LIN {X 0,Y 351.682,Z 414.171,A -85,B 0,C 180,E1 -13752.555,E2 -13752.555} C_VEL
LIN {X 0,Y 350.66,Z 425.768,A -85,B 0,C 180,E1 -13753.703,E2 -13753.703} C_VEL
LIN {X 0,Y 349.719,Z 436.215,A -85,B 0,C 180,E1 -13755.003,E2 -13755.003} C_VEL
LIN {X 0,Y 348.835,Z 444.735,A -85,B 0,C 180,E1 -13756.305,E2 -13756.305} C_VEL
LIN {X 0,Y 347.83,Z 453.948,A -85,B 0,C 180,E1 -13758.046,E2 -13758.046} C_VEL
LIN {X 0,Y 347.155,Z 461.359,A -85,B 0,C 180,E1 -13759.795,E2 -13759.795} C_VEL
LIN {X 0,Y 346.719,Z 466.377,A -85,B 0,C 180,E1 -13761.254,E2 -13761.254} C_VEL
LIN {X 0,Y 346.356,Z 471.237,A -85,B 0,C 180,E1 -13763.005,E2 -13763.005} C_VEL
LIN {X 0,Y 346.195,Z 474.523,A -85,B 0,C 180,E1 -13764.52,E2 -13764.52} C_VEL
LIN {X 0,Y 346.13,Z 477.65,A -85,B 0,C 180,E1 -13766.506,E2 -13766.506} C_VEL
LIN {X 0,Y 346.055,Z 478.914,A -85,B 0,C 180,E1 -13767.67,E2 -13767.67} C_VEL
LIN {X 0,Y 346.058,Z 479.779,A -85,B 0,C 180,E1 -13768.835,E2 -13768.835} C_VEL
LIN {X 0,Y 346.083,Z 480.204,A -85,B 0,C 180,E1 -13769.998,E2 -13769.998} C_VEL
LIN {X 0,Y 346.056,Z 480.234,A -85,B 0,C 180,E1 -13771.162,E2 -13771.162} C_VEL
LIN {X 0,Y 346.135,Z 479.143,A -85,B 0,C 180,E1 -13773.49,E2 -13773.49} C_VEL
LIN {X 0,Y 346.218,Z 477.967,A -85,B 0,C 180,E1 -13774.656,E2 -13774.656} C_VEL
LIN {X 0,Y 346.439,Z 474.38,A -85,B 0,C 180,E1 -13776.989,E2 -13776.989} C_VEL
LIN {X 0,Y 346.874,Z 470.515,A -85,B 0,C 180,E1 -13778.738,E2 -13778.738} C_VEL
LIN {X 0,Y 347.491,Z 465.542,A -85,B 0,C 180,E1 -13780.486,E2 -13780.486} C_VEL
LIN {X 0,Y 348.32,Z 459.311,A -85,B 0,C 180,E1 -13782.229,E2 -13782.229} C_VEL
LIN {X 0,Y 349.563,Z 451.533,A -85,B 0,C 180,E1 -13783.959,E2 -13783.959} C_VEL
LIN {X 0,Y 350.816,Z 442.76,A -85,B 0,C 180,E1 -13785.536,E2 -13785.536} C_VEL
LIN {X 0,Y 352.063,Z 433.253,A -85,B 0,C 180,E1 -13786.928,E2 -13786.928} C_VEL
LIN {X 0,Y 353.417,Z 423.319,A -85,B 0,C 180,E1 -13788.1,E2 -13788.1} C_VEL
LIN {X 0,Y 354.601,Z 412.984,A -85,B 0,C 180,E1 -13789.086,E2 -13789.086} C_VEL
LIN {X 0,Y 355.85,Z 400.601,A -85,B 0,C 180,E1 -13789.992,E2 -13789.992} C_VEL
LIN {X 0,Y 356.855,Z 387.621,A -85,B 0,C 180,E1 -13790.685,E2 -13790.685} C_VEL
LIN {X 0,Y 357.633,Z 374.787,A -85,B 0,C 180,E1 -13791.128,E2 -13791.128} C_VEL
LIN {X 0,Y 359.147,Z 301.824,A -85,B 0,C 180,E1 -13792.662,E2 -13792.662} C_VEL
LIN {X 0,Y 355.404,Z 281.679,A -85,B 0,C 180,E1 -13793.422,E2 -13793.422} C_VEL
LIN {X 0,Y 352.356,Z 268.39,A -85,B 0,C 180,E1 -13794.005,E2 -13794.005} C_VEL
LIN {X 0,Y 352.467,Z 266.171,A -85,B 0,C 180,E1 -13794.469,E2 -13794.469} C_VEL
LIN {X 0,Y 351.097,Z 258.022,A -85,B 0,C 180,E1 -13796.766,E2 -13796.766} C_VEL
LIN {X 0,Y 348.703,Z 247.494,A -85,B 0,C 180,E1 -13799.923,E2 -13799.923} C_VEL
LIN {X 0,Y 347.77,Z 243.712,A -85,B 0,C 180,E1 -13801.186,E2 -13801.186} C_VEL
LIN {X 0,Y 347.749,Z 243.664,A -85,B 0,C 180,E1 -13804.461,E2 -13804.461} C_VEL
LIN {X 0,Y 347.768,Z 243.657,A -85,B 0,C 180,E1 -13807.983,E2 -13807.983} C_VEL
LIN {X 0,Y 347.75,Z 243.656,A -85,B 0,C 180,E1 -13811.827,E2 -13811.827} C_VEL
LIN {X 0,Y 347.707,Z 243.67,A -85,B 0,C 180,E1 -13815.024,E2 -13815.024} C_VEL
LIN {X 0,Y 347.742,Z 243.664,A -85,B 0,C 180,E1 -13818.395,E2 -13818.395} C_VEL
LIN {X 0,Y 347.756,Z 243.666,A -85,B 0,C 180,E1 -13822.675,E2 -13822.675} C_VEL
LIN {X 0,Y 347.748,Z 243.668,A -85,B 0,C 180,E1 -13825.952,E2 -13825.952} C_VEL
LIN {X 0,Y 347.736,Z 243.667,A -85,B 0,C 180,E1 -13829.647,E2 -13829.647} C_VEL
LIN {X 0,Y 347.741,Z 243.665,A -85,B 0,C 180,E1 -13833.597,E2 -13833.597} C_VEL
LIN {X 0,Y 347.745,Z 243.665,A -85,B 0,C 180,E1 -13836.155,E2 -13836.155} C_VEL
LIN {X 0,Y 347.792,Z 243.658,A -85,B 0,C 180,E1 -13839.904,E2 -13839.904} C_VEL
LIN {X 0,Y 347.824,Z 243.651,A -85,B 0,C 180,E1 -13843.564,E2 -13843.564} C_VEL
LIN {X 0,Y 347.88,Z 243.644,A -85,B 0,C 180,E1 -13847.156,E2 -13847.156} C_VEL
LIN {X 0,Y 347.924,Z 243.645,A -85,B 0,C 180,E1 -13850.696,E2 -13850.696} C_VEL
LIN {X 0,Y 348.057,Z 243.62,A -85,B 0,C 180,E1 -13853.037,E2 -13853.037} C_VEL
LIN {X 0,Y 348.167,Z 243.61,A -85,B 0,C 180,E1 -13857.682,E2 -13857.682} C_VEL
LIN {X 0,Y 348.101,Z 243.616,A -85,B 0,C 180,E1 -13861.152,E2 -13861.152} C_VEL
LIN {X 0,Y 348.174,Z 243.612,A -85,B 0,C 180,E1 -13862.309,E2 -13862.309} C_VEL
LIN {X 0,Y 348.034,Z 243.629,A -85,B 0,C 180,E1 -13866.954,E2 -13866.954} C_VEL
LIN {X 0,Y 347.877,Z 243.65,A -85,B 0,C 180,E1 -13870.471,E2 -13870.471} C_VEL
LIN {X 0,Y 347.878,Z 243.65,A -85,B 0,C 180,E1 -13874.146,E2 -13874.146} C_VEL
LIN {X 0,Y 347.806,Z 243.662,A -85,B 0,C 180,E1 -13878.255,E2 -13878.255} C_VEL
LIN {X 0,Y 347.743,Z 243.669,A -85,B 0,C 180,E1 -13881.622,E2 -13881.622} C_VEL
LIN {X 0,Y 347.784,Z 243.658,A -85,B 0,C 180,E1 -13885.105,E2 -13885.105} C_VEL
LIN {X 0,Y 347.78,Z 243.657,A -85,B 0,C 180,E1 -13887.69,E2 -13887.69} C_VEL
LIN {X 0,Y 347.72,Z 243.671,A -85,B 0,C 180,E1 -13890.344,E2 -13890.344} C_VEL
LIN {X 0,Y 347.718,Z 243.672,A -85,B 0,C 180,E1 -13894.04,E2 -13894.04} C_VEL
LIN {X 0,Y 347.734,Z 243.671,A -85,B 0,C 180,E1 -13897.317,E2 -13897.317} C_VEL
LIN {X 0,Y 347.795,Z 243.745,A -85,B 0,C 180,E1 -13900.143,E2 -13900.143} C_VEL
LIN {X 0,Y 349.721,Z 251.799,A -85,B 0,C 180,E1 -13902.698,E2 -13902.698} C_VEL
LIN {X 0,Y 351.322,Z 259.614,A -85,B 0,C 180,E1 -13904.917,E2 -13904.917} C_VEL
LIN {X 0,Y 354.745,Z 268.202,A -85,B 0,C 180,E1 -13905.452,E2 -13905.452} C_VEL
LIN {X 0,Y 359.039,Z 287.558,A -85,B 0,C 180,E1 -13906.246,E2 -13906.246} C_VEL
LIN {X 0,Y 359.451,Z 290.704,A -85,B 0,C 180,E1 -13906.35,E2 -13906.35} C_VEL
LIN {X 0,Y 357.669,Z 366.827,A -85,B 0,C 180,E1 -13907.943,E2 -13907.943} C_VEL
LIN {X 0,Y 356.966,Z 380.05,A -85,B 0,C 180,E1 -13908.434,E2 -13908.434} C_VEL
LIN {X 0,Y 356.033,Z 392.461,A -85,B 0,C 180,E1 -13909.12,E2 -13909.12} C_VEL
LIN {X 0,Y 354.972,Z 403.655,A -85,B 0,C 180,E1 -13909.952,E2 -13909.952} C_VEL
LIN {X 0,Y 353.647,Z 415.17,A -85,B 0,C 180,E1 -13911.065,E2 -13911.065} C_VEL
LIN {X 0,Y 352.238,Z 425.645,A -85,B 0,C 180,E1 -13912.338,E2 -13912.338} C_VEL
LIN {X 0,Y 350.892,Z 435.215,A -85,B 0,C 180,E1 -13913.785,E2 -13913.785} C_VEL
LIN {X 0,Y 349.601,Z 444.237,A -85,B 0,C 180,E1 -13915.498,E2 -13915.498} C_VEL
LIN {X 0,Y 348.467,Z 451.785,A -85,B 0,C 180,E1 -13917.289,E2 -13917.289} C_VEL
LIN {X 0,Y 347.673,Z 457.456,A -85,B 0,C 180,E1 -13918.974,E2 -13918.974} C_VEL
LIN {X 0,Y 347.011,Z 462.595,A -85,B 0,C 180,E1 -13920.92,E2 -13920.92} C_VEL
LIN {X 0,Y 346.434,Z 466.863,A -85,B 0,C 180,E1 -13923.189,E2 -13923.189} C_VEL
LIN {X 0,Y 346.107,Z 468.889,A -85,B 0,C 180,E1 -13924.761,E2 -13924.761} C_VEL
LIN {X 0,Y 345.949,Z 469.985,A -85,B 0,C 180,E1 -13926.073,E2 -13926.073} C_VEL
LIN {X 0,Y 345.838,Z 470.579,A -85,B 0,C 180,E1 -13927.289,E2 -13927.289} C_VEL
LIN {X 0,Y 345.853,Z 470.615,A -85,B 0,C 180,E1 -13929.17,E2 -13929.17} C_VEL
LIN {X 0,Y 345.864,Z 469.63,A -85,B 0,C 180,E1 -13931.029,E2 -13931.029} C_VEL
LIN {X 0,Y 345.995,Z 467.897,A -85,B 0,C 180,E1 -13932.663,E2 -13932.663} C_VEL
LIN {X 0,Y 346.291,Z 464.592,A -85,B 0,C 180,E1 -13934.704,E2 -13934.704} C_VEL
LIN {X 0,Y 346.65,Z 460.054,A -85,B 0,C 180,E1 -13936.664,E2 -13936.664} C_VEL
LIN {X 0,Y 347.185,Z 454.043,A -85,B 0,C 180,E1 -13938.619,E2 -13938.619} C_VEL
LIN {X 0,Y 347.801,Z 447.067,A -85,B 0,C 180,E1 -13940.405,E2 -13940.405} C_VEL
LIN {X 0,Y 348.578,Z 439.91,A -85,B 0,C 180,E1 -13941.888,E2 -13941.888} C_VEL
LIN {X 0,Y 349.45,Z 431.284,A -85,B 0,C 180,E1 -13943.361,E2 -13943.361} C_VEL
LIN {X 0,Y 350.398,Z 421.777,A -85,B 0,C 180,E1 -13944.679,E2 -13944.679} C_VEL
LIN {X 0,Y 351.538,Z 409.922,A -85,B 0,C 180,E1 -13945.99,E2 -13945.99} C_VEL
LIN {X 0,Y 352.473,Z 398.031,A -85,B 0,C 180,E1 -13947.013,E2 -13947.013} C_VEL
LIN {X 0,Y 353.204,Z 386.003,A -85,B 0,C 180,E1 -13947.792,E2 -13947.792} C_VEL
LIN {X 0,Y 353.922,Z 372.608,A -85,B 0,C 180,E1 -13948.402,E2 -13948.402} C_VEL
LIN {X 0,Y 354.254,Z 359.778,A -85,B 0,C 180,E1 -13948.758,E2 -13948.758} C_VEL
LIN {X 0,Y 355.381,Z 287.662,A -85,B 0,C 180,E1 -13950.237,E2 -13950.237} C_VEL
LIN {X 0,Y 350.634,Z 259.687,A -85,B 0,C 180,E1 -13951.121,E2 -13951.121} C_VEL
LIN {X 0,Y 350.475,Z 257.185,A -85,B 0,C 180,E1 -13951.725,E2 -13951.725} C_VEL
LIN {X 0,Y 349.083,Z 250.011,A -85,B 0,C 180,E1 -13953.753,E2 -13953.753} C_VEL
LIN {X 0,Y 348.017,Z 243.683,A -85,B 0,C 180,E1 -13955.652,E2 -13955.652} C_VEL
LIN {X 0,Y 348.004,Z 243.633,A -85,B 0,C 180,E1 -13958.332,E2 -13958.332} C_VEL
LIN {X 0,Y 347.85,Z 243.658,A -85,B 0,C 180,E1 -13961.658,E2 -13961.658} C_VEL
LIN {X 0,Y 347.828,Z 243.656,A -85,B 0,C 180,E1 -13965.23,E2 -13965.23} C_VEL
LIN {X 0,Y 347.829,Z 243.654,A -85,B 0,C 180,E1 -13968.606,E2 -13968.606} C_VEL
LIN {X 0,Y 347.11,Z 243.749,A -85,B 0,C 180,E1 -13969.572,E2 -13969.572} C_VEL
LIN {X 0,Y 344.197,Z 244.107,A -85,B 0,C 180,E1 -13971.143,E2 -13971.143} C_VEL
LIN {X 0,Y 341.764,Z 244.411,A -85,B 0,C 180,E1 -13972.414,E2 -13972.414} C_VEL
LIN {X 0,Y 340.735,Z 244.539,A -85,B 0,C 180,E1 -13973.399,E2 -13973.399} C_VEL
LIN {X 0,Y 340.658,Z 244.546,A -85,B 0,C 180,E1 -13973.733,E2 -13973.733} C_VEL
LIN {X 0,Y 340.667,Z 244.547,A -85,B 0,C 180,E1 -13977.504,E2 -13977.504} C_VEL
LIN {X 0,Y 340.661,Z 244.547,A -85,B 0,C 180,E1 -13981.05,E2 -13981.05} C_VEL
LIN {X 0,Y 340.688,Z 244.544,A -85,B 0,C 180,E1 -13985.284,E2 -13985.284} C_VEL
LIN {X 0,Y 340.668,Z 244.552,A -85,B 0,C 180,E1 -13988.387,E2 -13988.387} C_VEL
LIN {X 0,Y 340.667,Z 244.547,A -85,B 0,C 180,E1 -13992.049,E2 -13992.049} C_VEL
LIN {X 0,Y 340.63,Z 244.552,A -85,B 0,C 180,E1 -13996.233,E2 -13996.233} C_VEL
LIN {X 0,Y 340.653,Z 244.552,A -85,B 0,C 180,E1 -13998.694,E2 -13998.694} C_VEL
LIN {X 0,Y 340.702,Z 244.541,A -85,B 0,C 180,E1 -14001.776,E2 -14001.776} C_VEL
LIN {X 0,Y 340.709,Z 244.542,A -85,B 0,C 180,E1 -14005.601,E2 -14005.601} C_VEL
LIN {X 0,Y 340.679,Z 244.548,A -85,B 0,C 180,E1 -14008.96,E2 -14008.96} C_VEL
LIN {X 0,Y 340.701,Z 244.544,A -85,B 0,C 180,E1 -14013.017,E2 -14013.017} C_VEL
LIN {X 0,Y 340.699,Z 244.544,A -85,B 0,C 180,E1 -14016.931,E2 -14016.931} C_VEL
LIN {X 0,Y 340.724,Z 244.538,A -85,B 0,C 180,E1 -14020.735,E2 -14020.735} C_VEL
LIN {X 0,Y 340.816,Z 244.526,A -85,B 0,C 180,E1 -14024.456,E2 -14024.456} C_VEL
LIN {X 0,Y 340.847,Z 244.527,A -85,B 0,C 180,E1 -14028.106,E2 -14028.106} C_VEL
LIN {X 0,Y 340.984,Z 244.511,A -85,B 0,C 180,E1 -14031.71,E2 -14031.71} C_VEL
LIN {X 0,Y 341.016,Z 244.506,A -85,B 0,C 180,E1 -14034.09,E2 -14034.09} C_VEL
LIN {X 0,Y 341.131,Z 244.488,A -85,B 0,C 180,E1 -14037.643,E2 -14037.643} C_VEL
LIN {X 0,Y 341.114,Z 244.49,A -85,B 0,C 180,E1 -14041.185,E2 -14041.185} C_VEL
LIN {X 0,Y 341.125,Z 244.494,A -85,B 0,C 180,E1 -14042.366,E2 -14042.366} C_VEL
LIN {X 0,Y 341.021,Z 244.504,A -85,B 0,C 180,E1 -14045.919,E2 -14045.919} C_VEL
LIN {X 0,Y 340.975,Z 244.512,A -85,B 0,C 180,E1 -14048.36,E2 -14048.36} C_VEL
LIN {X 0,Y 340.86,Z 244.522,A -85,B 0,C 180,E1 -14051.903,E2 -14051.903} C_VEL
LIN {X 0,Y 340.831,Z 244.526,A -85,B 0,C 180,E1 -14055.553,E2 -14055.553} C_VEL
LIN {X 0,Y 340.75,Z 244.536,A -85,B 0,C 180,E1 -14059.273,E2 -14059.273} C_VEL
LIN {X 0,Y 340.726,Z 244.543,A -85,B 0,C 180,E1 -14063.077,E2 -14063.077} C_VEL
LIN {X 0,Y 340.731,Z 244.539,A -85,B 0,C 180,E1 -14065.672,E2 -14065.672} C_VEL
LIN {X 0,Y 340.721,Z 244.54,A -85,B 0,C 180,E1 -14069.677,E2 -14069.677} C_VEL
LIN {X 0,Y 340.703,Z 244.542,A -85,B 0,C 180,E1 -14072.438,E2 -14072.438} C_VEL
LIN {X 0,Y 340.734,Z 244.544,A -85,B 0,C 180,E1 -14075.281,E2 -14075.281} C_VEL
LIN {X 0,Y 340.711,Z 244.54,A -85,B 0,C 180,E1 -14078.384,E2 -14078.384} C_VEL
LIN {X 0,Y 340.708,Z 244.542,A -85,B 0,C 180,E1 -14082.045,E2 -14082.045} C_VEL
LIN {X 0,Y 340.666,Z 244.547,A -85,B 0,C 180,E1 -14086.229,E2 -14086.229} C_VEL
LIN {X 0,Y 340.685,Z 244.544,A -85,B 0,C 180,E1 -14088.688,E2 -14088.688} C_VEL
LIN {X 0,Y 340.736,Z 244.543,A -85,B 0,C 180,E1 -14091.771,E2 -14091.771} C_VEL
LIN {X 0,Y 340.741,Z 244.54,A -85,B 0,C 180,E1 -14095.596,E2 -14095.596} C_VEL
LIN {X 0,Y 340.711,Z 244.545,A -85,B 0,C 180,E1 -14098.955,E2 -14098.955} C_VEL
LIN {X 0,Y 340.821,Z 244.72,A -85,B 0,C 180,E1 -14101.097,E2 -14101.097} C_VEL
LIN {X 0,Y 342.761,Z 254.35,A -85,B 0,C 180,E1 -14103.839,E2 -14103.839} C_VEL
LIN {X 0,Y 344.007,Z 261.845,A -85,B 0,C 180,E1 -14105.882,E2 -14105.882} C_VEL
LIN {X 0,Y 343.465,Z 268.458,A -85,B 0,C 180,E1 -14107.507,E2 -14107.507} C_VEL
LIN {X 0,Y 345.978,Z 284.64,A -85,B 0,C 180,E1 -14108.044,E2 -14108.044} C_VEL
LIN {X 0,Y 348.648,Z 302.169,A -85,B 0,C 180,E1 -14108.569,E2 -14108.569} C_VEL
LIN {X 0,Y 347.217,Z 376.561,A -85,B 0,C 180,E1 -14110.142,E2 -14110.142} C_VEL
LIN {X 0,Y 346.616,Z 389.671,A -85,B 0,C 180,E1 -14110.645,E2 -14110.645} C_VEL
LIN {X 0,Y 345.823,Z 401.785,A -85,B 0,C 180,E1 -14111.331,E2 -14111.331} C_VEL
LIN {X 0,Y 344.853,Z 413.215,A -85,B 0,C 180,E1 -14112.198,E2 -14112.198} C_VEL
LIN {X 0,Y 343.782,Z 424.984,A -85,B 0,C 180,E1 -14113.367,E2 -14113.367} C_VEL
LIN {X 0,Y 342.86,Z 435.072,A -85,B 0,C 180,E1 -14114.627,E2 -14114.627} C_VEL
LIN {X 0,Y 341.86,Z 444.184,A -85,B 0,C 180,E1 -14116.02,E2 -14116.02} C_VEL
LIN {X 0,Y 341.022,Z 452.127,A -85,B 0,C 180,E1 -14117.501,E2 -14117.501} C_VEL
LIN {X 0,Y 340.243,Z 459.861,A -85,B 0,C 180,E1 -14119.284,E2 -14119.284} C_VEL
LIN {X 0,Y 339.69,Z 466.063,A -85,B 0,C 180,E1 -14121.072,E2 -14121.072} C_VEL
LIN {X 0,Y 339.288,Z 470.97,A -85,B 0,C 180,E1 -14122.859,E2 -14122.859} C_VEL
LIN {X 0,Y 339.09,Z 474.652,A -85,B 0,C 180,E1 -14124.6,E2 -14124.6} C_VEL
LIN {X 0,Y 339.056,Z 477.469,A -85,B 0,C 180,E1 -14126.433,E2 -14126.433} C_VEL
LIN {X 0,Y 338.964,Z 479.638,A -85,B 0,C 180,E1 -14128.81,E2 -14128.81} C_VEL
LIN {X 0,Y 338.986,Z 480.095,A -85,B 0,C 180,E1 -14129.998,E2 -14129.998} C_VEL
LIN {X 0,Y 338.971,Z 479.811,A -85,B 0,C 180,E1 -14132.375,E2 -14132.375} C_VEL
LIN {X 0,Y 339.064,Z 479.095,A -85,B 0,C 180,E1 -14133.563,E2 -14133.563} C_VEL
LIN {X 0,Y 339.119,Z 477.959,A -85,B 0,C 180,E1 -14134.753,E2 -14134.753} C_VEL
LIN {X 0,Y 339.37,Z 474.421,A -85,B 0,C 180,E1 -14137.136,E2 -14137.136} C_VEL
LIN {X 0,Y 339.851,Z 470.604,A -85,B 0,C 180,E1 -14138.92,E2 -14138.92} C_VEL
LIN {X 0,Y 340.488,Z 465.68,A -85,B 0,C 180,E1 -14140.704,E2 -14140.704} C_VEL
LIN {X 0,Y 341.377,Z 459.504,A -85,B 0,C 180,E1 -14142.482,E2 -14142.482} C_VEL
LIN {X 0,Y 342.683,Z 451.821,A -85,B 0,C 180,E1 -14144.245,E2 -14144.245} C_VEL
LIN {X 0,Y 343.951,Z 443.371,A -85,B 0,C 180,E1 -14145.812,E2 -14145.812} C_VEL
LIN {X 0,Y 345.345,Z 433.39,A -85,B 0,C 180,E1 -14147.313,E2 -14147.313} C_VEL
LIN {X 0,Y 346.846,Z 422.594,A -85,B 0,C 180,E1 -14148.609,E2 -14148.609} C_VEL
LIN {X 0,Y 348.37,Z 410.306,A -85,B 0,C 180,E1 -14149.748,E2 -14149.748} C_VEL
LIN {X 0,Y 349.521,Z 398.32,A -85,B 0,C 180,E1 -14150.6,E2 -14150.6} C_VEL
LIN {X 0,Y 350.521,Z 386.003,A -85,B 0,C 180,E1 -14151.23,E2 -14151.23} C_VEL
LIN {X 0,Y 351.237,Z 373.363,A -85,B 0,C 180,E1 -14151.647,E2 -14151.647} C_VEL
LIN {X 0,Y 352.787,Z 302.833,A -85,B 0,C 180,E1 -14153.151,E2 -14153.151} C_VEL
LIN {X 0,Y 349.123,Z 283.054,A -85,B 0,C 180,E1 -14153.922,E2 -14153.922} C_VEL
LIN {X 0,Y 345.671,Z 268.186,A -85,B 0,C 180,E1 -14154.609,E2 -14154.609} C_VEL
LIN {X 0,Y 345.341,Z 265.378,A -85,B 0,C 180,E1 -14155.298,E2 -14155.298} C_VEL
LIN {X 0,Y 343.273,Z 255.226,A -85,B 0,C 180,E1 -14158.309,E2 -14158.309} C_VEL
LIN {X 0,Y 340.746,Z 244.756,A -85,B 0,C 180,E1 -14161.643,E2 -14161.643} C_VEL
LIN {X 0,Y 340.723,Z 244.535,A -85,B 0,C 180,E1 -14165.276,E2 -14165.276} C_VEL
LIN {X 0,Y 340.698,Z 244.536,A -85,B 0,C 180,E1 -14168.379,E2 -14168.379} C_VEL
LIN {X 0,Y 340.699,Z 244.533,A -85,B 0,C 180,E1 -14172.041,E2 -14172.041} C_VEL
LIN {X 0,Y 340.653,Z 244.535,A -85,B 0,C 180,E1 -14176.224,E2 -14176.224} C_VEL
LIN {X 0,Y 340.673,Z 244.549,A -85,B 0,C 180,E1 -14178.684,E2 -14178.684} C_VEL
LIN {X 0,Y 340.719,Z 244.541,A -85,B 0,C 180,E1 -14181.767,E2 -14181.767} C_VEL
LIN {X 0,Y 340.723,Z 244.542,A -85,B 0,C 180,E1 -14185.592,E2 -14185.592} C_VEL
LIN {X 0,Y 340.692,Z 244.548,A -85,B 0,C 180,E1 -14188.951,E2 -14188.951} C_VEL
LIN {X 0,Y 340.715,Z 244.544,A -85,B 0,C 180,E1 -14193.008,E2 -14193.008} C_VEL
LIN {X 0,Y 340.697,Z 244.548,A -85,B 0,C 180,E1 -14196.921,E2 -14196.921} C_VEL
LIN {X 0,Y 340.728,Z 244.541,A -85,B 0,C 180,E1 -14200.726,E2 -14200.726} C_VEL
LIN {X 0,Y 340.81,Z 244.527,A -85,B 0,C 180,E1 -14204.446,E2 -14204.446} C_VEL
LIN {X 0,Y 340.838,Z 244.519,A -85,B 0,C 180,E1 -14208.096,E2 -14208.096} C_VEL
LIN {X 0,Y 340.97,Z 244.502,A -85,B 0,C 180,E1 -14211.7,E2 -14211.7} C_VEL
LIN {X 0,Y 341.011,Z 244.505,A -85,B 0,C 180,E1 -14214.081,E2 -14214.081} C_VEL
LIN {X 0,Y 341.103,Z 244.489,A -85,B 0,C 180,E1 -14217.634,E2 -14217.634} C_VEL
LIN {X 0,Y 341.072,Z 244.492,A -85,B 0,C 180,E1 -14221.176,E2 -14221.176} C_VEL
LIN {X 0,Y 341.111,Z 244.492,A -85,B 0,C 180,E1 -14222.357,E2 -14222.357} C_VEL
LIN {X 0,Y 340.982,Z 244.508,A -85,B 0,C 180,E1 -14227.099,E2 -14227.099} C_VEL
LIN {X 0,Y 340.828,Z 244.528,A -85,B 0,C 180,E1 -14230.69,E2 -14230.69} C_VEL
LIN {X 0,Y 340.843,Z 244.529,A -85,B 0,C 180,E1 -14234.32,E2 -14234.32} C_VEL
LIN {X 0,Y 340.763,Z 244.538,A -85,B 0,C 180,E1 -14238.436,E2 -14238.436} C_VEL
LIN {X 0,Y 340.693,Z 244.548,A -85,B 0,C 180,E1 -14241.837,E2 -14241.837} C_VEL
LIN {X 0,Y 340.745,Z 244.536,A -85,B 0,C 180,E1 -14245.66,E2 -14245.66} C_VEL
LIN {X 0,Y 340.7,Z 244.533,A -85,B 0,C 180,E1 -14248.317,E2 -14248.317} C_VEL
LIN {X 0,Y 340.668,Z 244.549,A -85,B 0,C 180,E1 -14251.041,E2 -14251.041} C_VEL
LIN {X 0,Y 340.687,Z 244.541,A -85,B 0,C 180,E1 -14255.275,E2 -14255.275} C_VEL
LIN {X 0,Y 340.719,Z 244.558,A -85,B 0,C 180,E1 -14259.466,E2 -14259.466} C_VEL
LIN {X 0,Y 340.766,Z 244.925,A -85,B 0,C 180,E1 -14259.735,E2 -14259.735} C_VEL
LIN {X 0,Y 342.942,Z 253.734,A -85,B 0,C 180,E1 -14262.545,E2 -14262.545} C_VEL
LIN {X 0,Y 344.15,Z 259.548,A -85,B 0,C 180,E1 -14264.242,E2 -14264.242} C_VEL
LIN {X 0,Y 345.966,Z 263.998,A -85,B 0,C 180,E1 -14264.579,E2 -14264.579} C_VEL
LIN {X 0,Y 348.905,Z 271.265,A -85,B 0,C 180,E1 -14265.018,E2 -14265.018} C_VEL
LIN {X 0,Y 353.009,Z 290.5,A -85,B 0,C 180,E1 -14265.821,E2 -14265.821} C_VEL
LIN {X 0,Y 351.219,Z 367.472,A -85,B 0,C 180,E1 -14267.475,E2 -14267.475} C_VEL
LIN {X 0,Y 350.475,Z 380.66,A -85,B 0,C 180,E1 -14267.981,E2 -14267.981} C_VEL
LIN {X 0,Y 349.468,Z 393.467,A -85,B 0,C 180,E1 -14268.712,E2 -14268.712} C_VEL
LIN {X 0,Y 348.301,Z 404.837,A -85,B 0,C 180,E1 -14269.596,E2 -14269.596} C_VEL
LIN {X 0,Y 346.843,Z 416.723,A -85,B 0,C 180,E1 -14270.794,E2 -14270.794} C_VEL
LIN {X 0,Y 345.31,Z 427.619,A -85,B 0,C 180,E1 -14272.187,E2 -14272.187} C_VEL
LIN {X 0,Y 343.92,Z 436.784,A -85,B 0,C 180,E1 -14273.66,E2 -14273.66} C_VEL
LIN {X 0,Y 342.607,Z 445.314,A -85,B 0,C 180,E1 -14275.357,E2 -14275.357} C_VEL
LIN {X 0,Y 341.58,Z 451.862,A -85,B 0,C 180,E1 -14276.962,E2 -14276.962} C_VEL
LIN {X 0,Y 340.605,Z 458.337,A -85,B 0,C 180,E1 -14278.948,E2 -14278.948} C_VEL
LIN {X 0,Y 339.933,Z 463.249,A -85,B 0,C 180,E1 -14280.934,E2 -14280.934} C_VEL
LIN {X 0,Y 339.42,Z 466.837,A -85,B 0,C 180,E1 -14282.903,E2 -14282.903} C_VEL
LIN {X 0,Y 339.103,Z 468.567,A -85,B 0,C 180,E1 -14284.202,E2 -14284.202} C_VEL
LIN {X 0,Y 338.858,Z 470.027,A -85,B 0,C 180,E1 -14285.847,E2 -14285.847} C_VEL
LIN {X 0,Y 338.71,Z 470.817,A -85,B 0,C 180,E1 -14288.071,E2 -14288.071} C_VEL
LIN {X 0,Y 338.769,Z 470.635,A -85,B 0,C 180,E1 -14289.351,E2 -14289.351} C_VEL
LIN {X 0,Y 338.741,Z 469.991,A -85,B 0,C 180,E1 -14290.614,E2 -14290.614} C_VEL
LIN {X 0,Y 338.88,Z 468.164,A -85,B 0,C 180,E1 -14292.529,E2 -14292.529} C_VEL
LIN {X 0,Y 339.141,Z 465.37,A -85,B 0,C 180,E1 -14294.374,E2 -14294.374} C_VEL
LIN {X 0,Y 339.475,Z 461.576,A -85,B 0,C 180,E1 -14296.178,E2 -14296.178} C_VEL
LIN {X 0,Y 339.912,Z 456.356,A -85,B 0,C 180,E1 -14298.069,E2 -14298.069} C_VEL
LIN {X 0,Y 340.495,Z 449.935,A -85,B 0,C 180,E1 -14299.897,E2 -14299.897} C_VEL
LIN {X 0,Y 341.332,Z 441.852,A -85,B 0,C 180,E1 -14301.715,E2 -14301.715} C_VEL
LIN {X 0,Y 342.261,Z 433.569,A -85,B 0,C 180,E1 -14303.221,E2 -14303.221} C_VEL
LIN {X 0,Y 343.271,Z 423.48,A -85,B 0,C 180,E1 -14304.716,E2 -14304.716} C_VEL
LIN {X 0,Y 344.353,Z 413.456,A -85,B 0,C 180,E1 -14305.906,E2 -14305.906} C_VEL
LIN {X 0,Y 345.364,Z 401.308,A -85,B 0,C 180,E1 -14307.044,E2 -14307.044} C_VEL
LIN {X 0,Y 346.194,Z 389.486,A -85,B 0,C 180,E1 -14307.893,E2 -14307.893} C_VEL
LIN {X 0,Y 346.878,Z 376.89,A -85,B 0,C 180,E1 -14308.551,E2 -14308.551} C_VEL
LIN {X 0,Y 347.312,Z 363.839,A -85,B 0,C 180,E1 -14308.987,E2 -14308.987} C_VEL
LIN {X 0,Y 348.621,Z 288.612,A -85,B 0,C 180,E1 -14310.566,E2 -14310.566} C_VEL
LIN {X 0,Y 343.737,Z 259.862,A -85,B 0,C 180,E1 -14311.496,E2 -14311.496} C_VEL
LIN {X 0,Y 343.166,Z 256.524,A -85,B 0,C 180,E1 -14312.349,E2 -14312.349} C_VEL
LIN {X 0,Y 341.026,Z 244.855,A -85,B 0,C 180,E1 -14315.768,E2 -14315.768} C_VEL
LIN {X 0,Y 340.998,Z 244.51,A -85,B 0,C 180,E1 -14316.214,E2 -14316.214} C_VEL
LIN {X 0,Y 340.876,Z 244.526,A -85,B 0,C 180,E1 -14319.496,E2 -14319.496} C_VEL
LIN {X 0,Y 340.809,Z 244.53,A -85,B 0,C 180,E1 -14323.113,E2 -14323.113} C_VEL
LIN {X 0,Y 340.75,Z 244.534,A -85,B 0,C 180,E1 -14326.785,E2 -14326.785} C_VEL
LIN {X 0,Y 340.753,Z 244.537,A -85,B 0,C 180,E1 -14329.27,E2 -14329.27} C_VEL
LIN {X 0,Y 340.67,Z 244.546,A -85,B 0,C 180,E1 -14333.079,E2 -14333.079} C_VEL
LIN {X 0,Y 340.658,Z 244.546,A -85,B 0,C 180,E1 -14333.733,E2 -14333.733} C_VEL
LIN {X 0,Y 339.999,Z 244.632,A -85,B 0,C 180,E1 -14334.719,E2 -14334.719} C_VEL
LIN {X 0,Y 337.119,Z 244.992,A -85,B 0,C 180,E1 -14336.323,E2 -14336.323} C_VEL
LIN {X 0,Y 334.693,Z 245.291,A -85,B 0,C 180,E1 -14337.622,E2 -14337.622} C_VEL
LIN {X 0,Y 333.685,Z 245.418,A -85,B 0,C 180,E1 -14338.627,E2 -14338.627} C_VEL
LIN {X 0,Y 333.621,Z 245.425,A -85,B 0,C 180,E1 -14338.968,E2 -14338.968} C_VEL
LIN {X 0,Y 333.612,Z 245.427,A -85,B 0,C 180,E1 -14342.591,E2 -14342.591} C_VEL
LIN {X 0,Y 333.646,Z 245.425,A -85,B 0,C 180,E1 -14346.145,E2 -14346.145} C_VEL
LIN {X 0,Y 333.577,Z 245.428,A -85,B 0,C 180,E1 -14349.204,E2 -14349.204} C_VEL
LIN {X 0,Y 333.604,Z 245.431,A -85,B 0,C 180,E1 -14352.504,E2 -14352.504} C_VEL
LIN {X 0,Y 333.574,Z 245.43,A -85,B 0,C 180,E1 -14355.96,E2 -14355.96} C_VEL
LIN {X 0,Y 333.585,Z 245.427,A -85,B 0,C 180,E1 -14359.33,E2 -14359.33} C_VEL
LIN {X 0,Y 333.646,Z 245.425,A -85,B 0,C 180,E1 -14363.175,E2 -14363.175} C_VEL
LIN {X 0,Y 333.659,Z 245.422,A -85,B 0,C 180,E1 -14365.347,E2 -14365.347} C_VEL
LIN {X 0,Y 333.615,Z 245.423,A -85,B 0,C 180,E1 -14368.227,E2 -14368.227} C_VEL
LIN {X 0,Y 333.618,Z 245.424,A -85,B 0,C 180,E1 -14371.026,E2 -14371.026} C_VEL
LIN {X 0,Y 333.65,Z 245.422,A -85,B 0,C 180,E1 -14374.928,E2 -14374.928} C_VEL
LIN {X 0,Y 333.654,Z 245.421,A -85,B 0,C 180,E1 -14379.023,E2 -14379.023} C_VEL
LIN {X 0,Y 333.738,Z 245.411,A -85,B 0,C 180,E1 -14381.592,E2 -14381.592} C_VEL
LIN {X 0,Y 333.808,Z 245.403,A -85,B 0,C 180,E1 -14385.582,E2 -14385.582} C_VEL
LIN {X 0,Y 333.815,Z 245.4,A -85,B 0,C 180,E1 -14389.083,E2 -14389.083} C_VEL
LIN {X 0,Y 333.959,Z 245.381,A -85,B 0,C 180,E1 -14392.751,E2 -14392.751} C_VEL
LIN {X 0,Y 333.781,Z 245.401,A -85,B 0,C 180,E1 -14395.174,E2 -14395.174} C_VEL
LIN {X 0,Y 334.071,Z 245.365,A -85,B 0,C 180,E1 -14397.593,E2 -14397.593} C_VEL
LIN {X 0,Y 334.082,Z 245.366,A -85,B 0,C 180,E1 -14401.21,E2 -14401.21} C_VEL
LIN {X 0,Y 334.065,Z 245.373,A -85,B 0,C 180,E1 -14402.416,E2 -14402.416} C_VEL
LIN {X 0,Y 333.995,Z 245.38,A -85,B 0,C 180,E1 -14406.044,E2 -14406.044} C_VEL
LIN {X 0,Y 333.924,Z 245.388,A -85,B 0,C 180,E1 -14408.476,E2 -14408.476} C_VEL
LIN {X 0,Y 333.802,Z 245.402,A -85,B 0,C 180,E1 -14412.159,E2 -14412.159} C_VEL
LIN {X 0,Y 333.822,Z 245.405,A -85,B 0,C 180,E1 -14414.638,E2 -14414.638} C_VEL
LIN {X 0,Y 333.739,Z 245.413,A -85,B 0,C 180,E1 -14418.621,E2 -14418.621} C_VEL
LIN {X 0,Y 333.668,Z 245.417,A -85,B 0,C 180,E1 -14422.284,E2 -14422.284} C_VEL
LIN {X 0,Y 333.703,Z 245.419,A -85,B 0,C 180,E1 -14425.092,E2 -14425.092} C_VEL
LIN {X 0,Y 333.668,Z 245.422,A -85,B 0,C 180,E1 -14428.98,E2 -14428.98} C_VEL
LIN {X 0,Y 333.661,Z 245.42,A -85,B 0,C 180,E1 -14432.589,E2 -14432.589} C_VEL
LIN {X 0,Y 333.692,Z 245.414,A -85,B 0,C 180,E1 -14436.141,E2 -14436.141} C_VEL
LIN {X 0,Y 333.637,Z 245.425,A -85,B 0,C 180,E1 -14439.198,E2 -14439.198} C_VEL
LIN {X 0,Y 333.643,Z 245.42,A -85,B 0,C 180,E1 -14442.5,E2 -14442.5} C_VEL
LIN {X 0,Y 333.61,Z 245.428,A -85,B 0,C 180,E1 -14445.955,E2 -14445.955} C_VEL
LIN {X 0,Y 333.619,Z 245.426,A -85,B 0,C 180,E1 -14449.326,E2 -14449.326} C_VEL
LIN {X 0,Y 333.68,Z 245.417,A -85,B 0,C 180,E1 -14453.169,E2 -14453.169} C_VEL
LIN {X 0,Y 333.692,Z 245.416,A -85,B 0,C 180,E1 -14455.341,E2 -14455.341} C_VEL
LIN {X 0,Y 333.647,Z 245.425,A -85,B 0,C 180,E1 -14458.222,E2 -14458.222} C_VEL
LIN {X 0,Y 333.742,Z 245.54,A -85,B 0,C 180,E1 -14460.77,E2 -14460.77} C_VEL
LIN {X 0,Y 336.013,Z 256.885,A -85,B 0,C 180,E1 -14464.083,E2 -14464.083} C_VEL
LIN {X 0,Y 336.983,Z 262.629,A -85,B 0,C 180,E1 -14465.674,E2 -14465.674} C_VEL
LIN {X 0,Y 336.591,Z 268.449,A -85,B 0,C 180,E1 -14467.124,E2 -14467.124} C_VEL
LIN {X 0,Y 341.893,Z 303.794,A -85,B 0,C 180,E1 -14468.24,E2 -14468.24} C_VEL
LIN {X 0,Y 340.422,Z 376.263,A -85,B 0,C 180,E1 -14469.807,E2 -14469.807} C_VEL
LIN {X 0,Y 339.801,Z 389.436,A -85,B 0,C 180,E1 -14470.32,E2 -14470.32} C_VEL
LIN {X 0,Y 338.985,Z 401.584,A -85,B 0,C 180,E1 -14471.018,E2 -14471.018} C_VEL
LIN {X 0,Y 337.898,Z 413.848,A -85,B 0,C 180,E1 -14471.976,E2 -14471.976} C_VEL
LIN {X 0,Y 336.799,Z 425.479,A -85,B 0,C 180,E1 -14473.169,E2 -14473.169} C_VEL
LIN {X 0,Y 335.863,Z 435.419,A -85,B 0,C 180,E1 -14474.447,E2 -14474.447} C_VEL
LIN {X 0,Y 334.765,Z 445.337,A -85,B 0,C 180,E1 -14476.027,E2 -14476.027} C_VEL
LIN {X 0,Y 333.712,Z 454.41,A -85,B 0,C 180,E1 -14477.841,E2 -14477.841} C_VEL
LIN {X 0,Y 333.002,Z 461.713,A -85,B 0,C 180,E1 -14479.664,E2 -14479.664} C_VEL
LIN {X 0,Y 332.485,Z 467.532,A -85,B 0,C 180,E1 -14481.489,E2 -14481.489} C_VEL
LIN {X 0,Y 332.172,Z 472.097,A -85,B 0,C 180,E1 -14483.316,E2 -14483.316} C_VEL
LIN {X 0,Y 331.981,Z 475.554,A -85,B 0,C 180,E1 -14485.141,E2 -14485.141} C_VEL
LIN {X 0,Y 331.962,Z 477.272,A -85,B 0,C 180,E1 -14486.357,E2 -14486.357} C_VEL
LIN {X 0,Y 331.891,Z 478.577,A -85,B 0,C 180,E1 -14487.571,E2 -14487.571} C_VEL
LIN {X 0,Y 331.872,Z 479.486,A -85,B 0,C 180,E1 -14488.785,E2 -14488.785} C_VEL
LIN {X 0,Y 331.892,Z 479.985,A -85,B 0,C 180,E1 -14489.998,E2 -14489.998} C_VEL
LIN {X 0,Y 331.891,Z 479.744,A -85,B 0,C 180,E1 -14492.425,E2 -14492.425} C_VEL
LIN {X 0,Y 331.972,Z 479.049,A -85,B 0,C 180,E1 -14493.639,E2 -14493.639} C_VEL
LIN {X 0,Y 332.083,Z 476.682,A -85,B 0,C 180,E1 -14495.89,E2 -14495.89} C_VEL
LIN {X 0,Y 332.454,Z 473.331,A -85,B 0,C 180,E1 -14497.896,E2 -14497.896} C_VEL
LIN {X 0,Y 333.011,Z 469.208,A -85,B 0,C 180,E1 -14499.718,E2 -14499.718} C_VEL
LIN {X 0,Y 334.001,Z 462.924,A -85,B 0,C 180,E1 -14501.837,E2 -14501.837} C_VEL
LIN {X 0,Y 335.075,Z 456.102,A -85,B 0,C 180,E1 -14503.646,E2 -14503.646} C_VEL
LIN {X 0,Y 336.581,Z 447.602,A -85,B 0,C 180,E1 -14505.438,E2 -14505.438} C_VEL
LIN {X 0,Y 337.845,Z 438.902,A -85,B 0,C 180,E1 -14506.93,E2 -14506.93} C_VEL
LIN {X 0,Y 339.453,Z 428.211,A -85,B 0,C 180,E1 -14508.403,E2 -14508.403} C_VEL
LIN {X 0,Y 340.954,Z 417.556,A -85,B 0,C 180,E1 -14509.568,E2 -14509.568} C_VEL
LIN {X 0,Y 342.174,Z 407.597,A -85,B 0,C 180,E1 -14510.434,E2 -14510.434} C_VEL
LIN {X 0,Y 343.276,Z 395.86,A -85,B 0,C 180,E1 -14511.228,E2 -14511.228} C_VEL
LIN {X 0,Y 344.33,Z 382.424,A -85,B 0,C 180,E1 -14511.867,E2 -14511.867} C_VEL
LIN {X 0,Y 344.962,Z 369,A -85,B 0,C 180,E1 -14512.258,E2 -14512.258} C_VEL
LIN {X 0,Y 346.493,Z 303.892,A -85,B 0,C 180,E1 -14513.662,E2 -14513.662} C_VEL
LIN {X 0,Y 342.812,Z 284.155,A -85,B 0,C 180,E1 -14514.464,E2 -14514.464} C_VEL
LIN {X 0,Y 339.39,Z 270.037,A -85,B 0,C 180,E1 -14515.129,E2 -14515.129} C_VEL
LIN {X 0,Y 338.605,Z 267.684,A -85,B 0,C 180,E1 -14515.327,E2 -14515.327} C_VEL
LIN {X 0,Y 336.841,Z 258.676,A -85,B 0,C 180,E1 -14517.992,E2 -14517.992} C_VEL
LIN {X 0,Y 334.587,Z 249.116,A -85,B 0,C 180,E1 -14521.042,E2 -14521.042} C_VEL
LIN {X 0,Y 333.671,Z 245.486,A -85,B 0,C 180,E1 -14522.331,E2 -14522.331} C_VEL
LIN {X 0,Y 333.68,Z 245.417,A -85,B 0,C 180,E1 -14526.136,E2 -14526.136} C_VEL
LIN {X 0,Y 333.637,Z 245.421,A -85,B 0,C 180,E1 -14529.191,E2 -14529.191} C_VEL
LIN {X 0,Y 333.634,Z 245.414,A -85,B 0,C 180,E1 -14532.496,E2 -14532.496} C_VEL
LIN {X 0,Y 333.597,Z 245.416,A -85,B 0,C 180,E1 -14535.951,E2 -14535.951} C_VEL
LIN {X 0,Y 333.604,Z 245.43,A -85,B 0,C 180,E1 -14539.321,E2 -14539.321} C_VEL
LIN {X 0,Y 333.663,Z 245.418,A -85,B 0,C 180,E1 -14543.165,E2 -14543.165} C_VEL
LIN {X 0,Y 333.674,Z 245.421,A -85,B 0,C 180,E1 -14545.337,E2 -14545.337} C_VEL
LIN {X 0,Y 333.628,Z 245.423,A -85,B 0,C 180,E1 -14548.218,E2 -14548.218} C_VEL
LIN {X 0,Y 333.65,Z 245.418,A -85,B 0,C 180,E1 -14551.018,E2 -14551.018} C_VEL
LIN {X 0,Y 333.662,Z 245.416,A -85,B 0,C 180,E1 -14555.081,E2 -14555.081} C_VEL
LIN {X 0,Y 333.657,Z 245.415,A -85,B 0,C 180,E1 -14559.014,E2 -14559.014} C_VEL
LIN {X 0,Y 333.735,Z 245.411,A -85,B 0,C 180,E1 -14561.582,E2 -14561.582} C_VEL
LIN {X 0,Y 333.801,Z 245.405,A -85,B 0,C 180,E1 -14565.572,E2 -14565.572} C_VEL
LIN {X 0,Y 333.806,Z 245.4,A -85,B 0,C 180,E1 -14569.073,E2 -14569.073} C_VEL
LIN {X 0,Y 333.955,Z 245.374,A -85,B 0,C 180,E1 -14572.742,E2 -14572.742} C_VEL
LIN {X 0,Y 333.767,Z 245.41,A -85,B 0,C 180,E1 -14575.164,E2 -14575.164} C_VEL
LIN {X 0,Y 334.044,Z 245.368,A -85,B 0,C 180,E1 -14577.584,E2 -14577.584} C_VEL
LIN {X 0,Y 334.043,Z 245.367,A -85,B 0,C 180,E1 -14581.201,E2 -14581.201} C_VEL
LIN {X 0,Y 334.051,Z 245.371,A -85,B 0,C 180,E1 -14582.407,E2 -14582.407} C_VEL
LIN {X 0,Y 333.94,Z 245.381,A -85,B 0,C 180,E1 -14586.458,E2 -14586.458} C_VEL
LIN {X 0,Y 333.801,Z 245.399,A -85,B 0,C 180,E1 -14589.692,E2 -14589.692} C_VEL
LIN {X 0,Y 333.776,Z 245.401,A -85,B 0,C 180,E1 -14593.387,E2 -14593.387} C_VEL
LIN {X 0,Y 333.696,Z 245.413,A -85,B 0,C 180,E1 -14597.143,E2 -14597.143} C_VEL
LIN {X 0,Y 333.665,Z 245.418,A -85,B 0,C 180,E1 -14599.689,E2 -14599.689} C_VEL
LIN {X 0,Y 333.643,Z 245.423,A -85,B 0,C 180,E1 -14603.586,E2 -14603.586} C_VEL
LIN {X 0,Y 333.708,Z 245.418,A -85,B 0,C 180,E1 -14606.242,E2 -14606.242} C_VEL
LIN {X 0,Y 333.662,Z 245.409,A -85,B 0,C 180,E1 -14608.97,E2 -14608.97} C_VEL
LIN {X 0,Y 333.613,Z 245.418,A -85,B 0,C 180,E1 -14612.583,E2 -14612.583} C_VEL
LIN {X 0,Y 333.646,Z 245.417,A -85,B 0,C 180,E1 -14616.135,E2 -14616.135} C_VEL
LIN {X 0,Y 333.688,Z 245.611,A -85,B 0,C 180,E1 -14619.057,E2 -14619.057} C_VEL
LIN {X 0,Y 335.92,Z 254.528,A -85,B 0,C 180,E1 -14622.02,E2 -14622.02} C_VEL
LIN {X 0,Y 337.087,Z 259.905,A -85,B 0,C 180,E1 -14623.605,E2 -14623.605} C_VEL
LIN {X 0,Y 342.794,Z 273.216,A -85,B 0,C 180,E1 -14624.508,E2 -14624.508} C_VEL
LIN {X 0,Y 346.673,Z 291.291,A -85,B 0,C 180,E1 -14625.292,E2 -14625.292} C_VEL
LIN {X 0,Y 344.951,Z 363.504,A -85,B 0,C 180,E1 -14626.858,E2 -14626.858} C_VEL
LIN {X 0,Y 344.343,Z 376.769,A -85,B 0,C 180,E1 -14627.302,E2 -14627.302} C_VEL
LIN {X 0,Y 343.421,Z 388.807,A -85,B 0,C 180,E1 -14627.919,E2 -14627.919} C_VEL
LIN {X 0,Y 342.292,Z 400.302,A -85,B 0,C 180,E1 -14628.734,E2 -14628.734} C_VEL
LIN {X 0,Y 340.843,Z 412.311,A -85,B 0,C 180,E1 -14629.846,E2 -14629.846} C_VEL
LIN {X 0,Y 339.442,Z 422.438,A -85,B 0,C 180,E1 -14631.034,E2 -14631.034} C_VEL
LIN {X 0,Y 337.974,Z 431.859,A -85,B 0,C 180,E1 -14632.398,E2 -14632.398} C_VEL
LIN {X 0,Y 336.65,Z 440.083,A -85,B 0,C 180,E1 -14633.863,E2 -14633.863} C_VEL
LIN {X 0,Y 335.373,Z 447.781,A -85,B 0,C 180,E1 -14635.544,E2 -14635.544} C_VEL
LIN {X 0,Y 334.375,Z 453.968,A -85,B 0,C 180,E1 -14637.205,E2 -14637.205} C_VEL
LIN {X 0,Y 333.542,Z 459.148,A -85,B 0,C 180,E1 -14638.923,E2 -14638.923} C_VEL
LIN {X 0,Y 332.835,Z 463.891,A -85,B 0,C 180,E1 -14640.947,E2 -14640.947} C_VEL
LIN {X 0,Y 332.38,Z 466.83,A -85,B 0,C 180,E1 -14642.617,E2 -14642.617} C_VEL
LIN {X 0,Y 331.891,Z 469.572,A -85,B 0,C 180,E1 -14644.946,E2 -14644.946} C_VEL
LIN {X 0,Y 331.713,Z 470.472,A -85,B 0,C 180,E1 -14646.264,E2 -14646.264} C_VEL
LIN {X 0,Y 331.631,Z 470.868,A -85,B 0,C 180,E1 -14647.578,E2 -14647.578} C_VEL
LIN {X 0,Y 331.64,Z 470.832,A -85,B 0,C 180,E1 -14648.886,E2 -14648.886} C_VEL
LIN {X 0,Y 331.642,Z 470.346,A -85,B 0,C 180,E1 -14650.182,E2 -14650.182} C_VEL
LIN {X 0,Y 331.765,Z 468.421,A -85,B 0,C 180,E1 -14652.391,E2 -14652.391} C_VEL
LIN {X 0,Y 332.096,Z 465.015,A -85,B 0,C 180,E1 -14654.663,E2 -14654.663} C_VEL
LIN {X 0,Y 332.447,Z 460.951,A -85,B 0,C 180,E1 -14656.555,E2 -14656.555} C_VEL
LIN {X 0,Y 333.033,Z 454.653,A -85,B 0,C 180,E1 -14658.745,E2 -14658.745} C_VEL
LIN {X 0,Y 333.697,Z 447.757,A -85,B 0,C 180,E1 -14660.608,E2 -14660.608} C_VEL
LIN {X 0,Y 334.666,Z 439.152,A -85,B 0,C 180,E1 -14662.46,E2 -14662.46} C_VEL
LIN {X 0,Y 335.696,Z 429.274,A -85,B 0,C 180,E1 -14664.144,E2 -14664.144} C_VEL
LIN {X 0,Y 336.838,Z 419.265,A -85,B 0,C 180,E1 -14665.514,E2 -14665.514} C_VEL
LIN {X 0,Y 337.953,Z 408.183,A -85,B 0,C 180,E1 -14666.727,E2 -14666.727} C_VEL
LIN {X 0,Y 338.918,Z 395.852,A -85,B 0,C 180,E1 -14667.774,E2 -14667.774} C_VEL
LIN {X 0,Y 339.724,Z 382.857,A -85,B 0,C 180,E1 -14668.594,E2 -14668.594} C_VEL
LIN {X 0,Y 340.362,Z 369.6,A -85,B 0,C 180,E1 -14669.151,E2 -14669.151} C_VEL
LIN {X 0,Y 340.811,Z 349.535,A -85,B 0,C 180,E1 -14669.633,E2 -14669.633} C_VEL
LIN {X 0,Y 341.907,Z 289.798,A -85,B 0,C 180,E1 -14670.9,E2 -14670.9} C_VEL
LIN {X 0,Y 337.026,Z 261.455,A -85,B 0,C 180,E1 -14671.814,E2 -14671.814} C_VEL
LIN {X 0,Y 336.509,Z 259.476,A -85,B 0,C 180,E1 -14671.985,E2 -14671.985} C_VEL
LIN {X 0,Y 334.627,Z 249.753,A -85,B 0,C 180,E1 -14674.821,E2 -14674.821} C_VEL
LIN {X 0,Y 333.983,Z 245.44,A -85,B 0,C 180,E1 -14676.193,E2 -14676.193} C_VEL
LIN {X 0,Y 333.814,Z 245.406,A -85,B 0,C 180,E1 -14679.698,E2 -14679.698} C_VEL
LIN {X 0,Y 333.757,Z 245.411,A -85,B 0,C 180,E1 -14683.395,E2 -14683.395} C_VEL
LIN {X 0,Y 333.71,Z 245.411,A -85,B 0,C 180,E1 -14687.15,E2 -14687.15} C_VEL
LIN {X 0,Y 333.696,Z 245.419,A -85,B 0,C 180,E1 -14689.695,E2 -14689.695} C_VEL
LIN {X 0,Y 333.608,Z 245.427,A -85,B 0,C 180,E1 -14693.726,E2 -14693.726} C_VEL
LIN {X 0,Y 333.637,Z 245.423,A -85,B 0,C 180,E1 -14697.61,E2 -14697.61} C_VEL
LIN {X 0,Y 333.621,Z 245.425,A -85,B 0,C 180,E1 -14698.968,E2 -14698.968} C_VEL
LIN {X 0,Y 333,Z 245.507,A -85,B 0,C 180,E1 -14699.976,E2 -14699.976} C_VEL
LIN {X 0,Y 330.155,Z 245.864,A -85,B 0,C 180,E1 -14701.615,E2 -14701.615} C_VEL
LIN {X 0,Y 327.711,Z 246.166,A -85,B 0,C 180,E1 -14702.943,E2 -14702.943} C_VEL
LIN {X 0,Y 326.656,Z 246.293,A -85,B 0,C 180,E1 -14703.971,E2 -14703.971} C_VEL
LIN {X 0,Y 326.569,Z 246.302,A -85,B 0,C 180,E1 -14704.32,E2 -14704.32} C_VEL
LIN {X 0,Y 326.596,Z 246.299,A -85,B 0,C 180,E1 -14707.242,E2 -14707.242} C_VEL
LIN {X 0,Y 326.519,Z 246.309,A -85,B 0,C 180,E1 -14711.129,E2 -14711.129} C_VEL
LIN {X 0,Y 326.537,Z 246.307,A -85,B 0,C 180,E1 -14713.532,E2 -14713.532} C_VEL
LIN {X 0,Y 326.554,Z 246.305,A -85,B 0,C 180,E1 -14717.035,E2 -14717.035} C_VEL
LIN {X 0,Y 326.565,Z 246.304,A -85,B 0,C 180,E1 -14721.391,E2 -14721.391} C_VEL
LIN {X 0,Y 326.604,Z 246.303,A -85,B 0,C 180,E1 -14724.858,E2 -14724.858} C_VEL
LIN {X 0,Y 326.595,Z 246.299,A -85,B 0,C 180,E1 -14727.461,E2 -14727.461} C_VEL
LIN {X 0,Y 326.568,Z 246.297,A -85,B 0,C 180,E1 -14730.339,E2 -14730.339} C_VEL
LIN {X 0,Y 326.587,Z 246.302,A -85,B 0,C 180,E1 -14733.14,E2 -14733.14} C_VEL
LIN {X 0,Y 326.587,Z 246.304,A -85,B 0,C 180,E1 -14737.216,E2 -14737.216} C_VEL
LIN {X 0,Y 326.669,Z 246.29,A -85,B 0,C 180,E1 -14741.199,E2 -14741.199} C_VEL
LIN {X 0,Y 326.763,Z 246.278,A -85,B 0,C 180,E1 -14745.439,E2 -14745.439} C_VEL
LIN {X 0,Y 326.757,Z 246.279,A -85,B 0,C 180,E1 -14748.844,E2 -14748.844} C_VEL
LIN {X 0,Y 326.916,Z 246.258,A -85,B 0,C 180,E1 -14752.594,E2 -14752.594} C_VEL
LIN {X 0,Y 326.75,Z 246.276,A -85,B 0,C 180,E1 -14755.069,E2 -14755.069} C_VEL
LIN {X 0,Y 327.015,Z 246.242,A -85,B 0,C 180,E1 -14757.541,E2 -14757.541} C_VEL
LIN {X 0,Y 327.05,Z 246.242,A -85,B 0,C 180,E1 -14761.236,E2 -14761.236} C_VEL
LIN {X 0,Y 326.745,Z 246.282,A -85,B 0,C 180,E1 -14763.704,E2 -14763.704} C_VEL
LIN {X 0,Y 326.95,Z 246.259,A -85,B 0,C 180,E1 -14766.175,E2 -14766.175} C_VEL
LIN {X 0,Y 326.794,Z 246.269,A -85,B 0,C 180,E1 -14769.911,E2 -14769.911} C_VEL
LIN {X 0,Y 326.772,Z 246.277,A -85,B 0,C 180,E1 -14773.689,E2 -14773.689} C_VEL
LIN {X 0,Y 326.678,Z 246.288,A -85,B 0,C 180,E1 -14777.533,E2 -14777.533} C_VEL
LIN {X 0,Y 326.63,Z 246.293,A -85,B 0,C 180,E1 -14781.46,E2 -14781.46} C_VEL
LIN {X 0,Y 326.649,Z 246.294,A -85,B 0,C 180,E1 -14785.491,E2 -14785.491} C_VEL
LIN {X 0,Y 326.632,Z 246.293,A -85,B 0,C 180,E1 -14789.666,E2 -14789.666} C_VEL
LIN {X 0,Y 326.634,Z 246.297,A -85,B 0,C 180,E1 -14792.948,E2 -14792.948} C_VEL
LIN {X 0,Y 326.629,Z 246.297,A -85,B 0,C 180,E1 -14795.522,E2 -14795.522} C_VEL
LIN {X 0,Y 326.604,Z 246.302,A -85,B 0,C 180,E1 -14799.223,E2 -14799.223} C_VEL
LIN {X 0,Y 326.589,Z 246.299,A -85,B 0,C 180,E1 -14802.972,E2 -14802.972} C_VEL
LIN {X 0,Y 326.589,Z 246.3,A -85,B 0,C 180,E1 -14807.03,E2 -14807.03} C_VEL
LIN {X 0,Y 326.589,Z 246.299,A -85,B 0,C 180,E1 -14810.782,E2 -14810.782} C_VEL
LIN {X 0,Y 326.629,Z 246.296,A -85,B 0,C 180,E1 -14814.48,E2 -14814.48} C_VEL
LIN {X 0,Y 326.626,Z 246.298,A -85,B 0,C 180,E1 -14817.456,E2 -14817.456} C_VEL
LIN {X 0,Y 326.692,Z 246.38,A -85,B 0,C 180,E1 -14820.44,E2 -14820.44} C_VEL
LIN {X 0,Y 327.428,Z 250.178,A -85,B 0,C 180,E1 -14821.652,E2 -14821.652} C_VEL
LIN {X 0,Y 329.207,Z 259.226,A -85,B 0,C 180,E1 -14824.28,E2 -14824.28} C_VEL
LIN {X 0,Y 330.028,Z 264.616,A -85,B 0,C 180,E1 -14825.798,E2 -14825.798} C_VEL
LIN {X 0,Y 329.716,Z 268.432,A -85,B 0,C 180,E1 -14826.719,E2 -14826.719} C_VEL
LIN {X 0,Y 335.102,Z 303.473,A -85,B 0,C 180,E1 -14827.86,E2 -14827.86} C_VEL
LIN {X 0,Y 333.633,Z 375.962,A -85,B 0,C 180,E1 -14829.458,E2 -14829.458} C_VEL
LIN {X 0,Y 332.989,Z 389.199,A -85,B 0,C 180,E1 -14829.981,E2 -14829.981} C_VEL
LIN {X 0,Y 332.066,Z 402.506,A -85,B 0,C 180,E1 -14830.768,E2 -14830.768} C_VEL
LIN {X 0,Y 330.948,Z 414.473,A -85,B 0,C 180,E1 -14831.744,E2 -14831.744} C_VEL
LIN {X 0,Y 329.819,Z 425.971,A -85,B 0,C 180,E1 -14832.961,E2 -14832.961} C_VEL
LIN {X 0,Y 328.865,Z 435.785,A -85,B 0,C 180,E1 -14834.263,E2 -14834.263} C_VEL
LIN {X 0,Y 327.805,Z 444.787,A -85,B 0,C 180,E1 -14835.724,E2 -14835.724} C_VEL
LIN {X 0,Y 326.75,Z 453.942,A -85,B 0,C 180,E1 -14837.577,E2 -14837.577} C_VEL
LIN {X 0,Y 325.976,Z 461.308,A -85,B 0,C 180,E1 -14839.439,E2 -14839.439} C_VEL
LIN {X 0,Y 325.425,Z 467.198,A -85,B 0,C 180,E1 -14841.303,E2 -14841.303} C_VEL
LIN {X 0,Y 325.088,Z 471.82,A -85,B 0,C 180,E1 -14843.169,E2 -14843.169} C_VEL
LIN {X 0,Y 324.896,Z 475.322,A -85,B 0,C 180,E1 -14845.034,E2 -14845.034} C_VEL
LIN {X 0,Y 324.87,Z 477.075,A -85,B 0,C 180,E1 -14846.277,E2 -14846.277} C_VEL
LIN {X 0,Y 324.813,Z 478.403,A -85,B 0,C 180,E1 -14847.518,E2 -14847.518} C_VEL
LIN {X 0,Y 324.784,Z 479.334,A -85,B 0,C 180,E1 -14848.758,E2 -14848.758} C_VEL
LIN {X 0,Y 324.801,Z 479.869,A -85,B 0,C 180,E1 -14849.998,E2 -14849.998} C_VEL
LIN {X 0,Y 324.783,Z 479.968,A -85,B 0,C 180,E1 -14851.238,E2 -14851.238} C_VEL
LIN {X 0,Y 324.882,Z 479.003,A -85,B 0,C 180,E1 -14853.719,E2 -14853.719} C_VEL
LIN {X 0,Y 325.006,Z 476.885,A -85,B 0,C 180,E1 -14855.869,E2 -14855.869} C_VEL
LIN {X 0,Y 325.42,Z 473.396,A -85,B 0,C 180,E1 -14858.068,E2 -14858.068} C_VEL
LIN {X 0,Y 326.009,Z 469.321,A -85,B 0,C 180,E1 -14859.929,E2 -14859.929} C_VEL
LIN {X 0,Y 327.014,Z 463.09,A -85,B 0,C 180,E1 -14862.093,E2 -14862.093} C_VEL
LIN {X 0,Y 328.198,Z 456.324,A -85,B 0,C 180,E1 -14863.938,E2 -14863.938} C_VEL
LIN {X 0,Y 329.759,Z 447.926,A -85,B 0,C 180,E1 -14865.765,E2 -14865.765} C_VEL
LIN {X 0,Y 331.084,Z 439.332,A -85,B 0,C 180,E1 -14867.286,E2 -14867.286} C_VEL
LIN {X 0,Y 332.748,Z 428.775,A -85,B 0,C 180,E1 -14868.788,E2 -14868.788} C_VEL
LIN {X 0,Y 334.324,Z 418.307,A -85,B 0,C 180,E1 -14869.972,E2 -14869.972} C_VEL
LIN {X 0,Y 335.825,Z 406.721,A -85,B 0,C 180,E1 -14870.999,E2 -14870.999} C_VEL
LIN {X 0,Y 337.007,Z 394.765,A -85,B 0,C 180,E1 -14871.804,E2 -14871.804} C_VEL
LIN {X 0,Y 338.012,Z 381.84,A -85,B 0,C 180,E1 -14872.419,E2 -14872.419} C_VEL
LIN {X 0,Y 338.693,Z 367.963,A -85,B 0,C 180,E1 -14872.814,E2 -14872.814} C_VEL
LIN {X 0,Y 340.183,Z 304.606,A -85,B 0,C 180,E1 -14874.211,E2 -14874.211} C_VEL
LIN {X 0,Y 336.483,Z 284.912,A -85,B 0,C 180,E1 -14875.039,E2 -14875.039} C_VEL
LIN {X 0,Y 333.584,Z 272.97,A -85,B 0,C 180,E1 -14875.621,E2 -14875.621} C_VEL
LIN {X 0,Y 331.444,Z 267.613,A -85,B 0,C 180,E1 -14876.029,E2 -14876.029} C_VEL
LIN {X 0,Y 329.831,Z 259.657,A -85,B 0,C 180,E1 -14878.452,E2 -14878.452} C_VEL
LIN {X 0,Y 327.489,Z 249.749,A -85,B 0,C 180,E1 -14881.717,E2 -14881.717} C_VEL
LIN {X 0,Y 326.627,Z 246.326,A -85,B 0,C 180,E1 -14882.998,E2 -14882.998} C_VEL
LIN {X 0,Y 326.631,Z 246.298,A -85,B 0,C 180,E1 -14887.044,E2 -14887.044} C_VEL
LIN {X 0,Y 326.589,Z 246.306,A -85,B 0,C 180,E1 -14890.206,E2 -14890.206} C_VEL
LIN {X 0,Y 326.564,Z 246.303,A -85,B 0,C 180,E1 -14893.522,E2 -14893.522} C_VEL
LIN {X 0,Y 326.575,Z 246.287,A -85,B 0,C 180,E1 -14897.025,E2 -14897.025} C_VEL
LIN {X 0,Y 326.572,Z 246.302,A -85,B 0,C 180,E1 -14900.778,E2 -14900.778} C_VEL
LIN {X 0,Y 326.611,Z 246.297,A -85,B 0,C 180,E1 -14904.476,E2 -14904.476} C_VEL
LIN {X 0,Y 326.607,Z 246.295,A -85,B 0,C 180,E1 -14907.451,E2 -14907.451} C_VEL
LIN {X 0,Y 326.614,Z 246.296,A -85,B 0,C 180,E1 -14910.332,E2 -14910.332} C_VEL
LIN {X 0,Y 326.599,Z 246.296,A -85,B 0,C 180,E1 -14914.504,E2 -14914.504} C_VEL
LIN {X 0,Y 326.609,Z 246.294,A -85,B 0,C 180,E1 -14918.538,E2 -14918.538} C_VEL
LIN {X 0,Y 326.657,Z 246.29,A -85,B 0,C 180,E1 -14922.466,E2 -14922.466} C_VEL
LIN {X 0,Y 326.751,Z 246.281,A -85,B 0,C 180,E1 -14926.31,E2 -14926.31} C_VEL
LIN {X 0,Y 326.773,Z 246.279,A -85,B 0,C 180,E1 -14930.088,E2 -14930.088} C_VEL
LIN {X 0,Y 326.939,Z 246.26,A -85,B 0,C 180,E1 -14933.825,E2 -14933.825} C_VEL
LIN {X 0,Y 326.988,Z 246.246,A -85,B 0,C 180,E1 -14937.532,E2 -14937.532} C_VEL
LIN {X 0,Y 327.013,Z 246.242,A -85,B 0,C 180,E1 -14941.227,E2 -14941.227} C_VEL
LIN {X 0,Y 326.737,Z 246.286,A -85,B 0,C 180,E1 -14943.695,E2 -14943.695} C_VEL
LIN {X 0,Y 326.903,Z 246.259,A -85,B 0,C 180,E1 -14946.446,E2 -14946.446} C_VEL
LIN {X 0,Y 326.764,Z 246.276,A -85,B 0,C 180,E1 -14949.903,E2 -14949.903} C_VEL
LIN {X 0,Y 326.739,Z 246.279,A -85,B 0,C 180,E1 -14953.681,E2 -14953.681} C_VEL
LIN {X 0,Y 326.641,Z 246.293,A -85,B 0,C 180,E1 -14957.525,E2 -14957.525} C_VEL
LIN {X 0,Y 326.61,Z 246.298,A -85,B 0,C 180,E1 -14960.132,E2 -14960.132} C_VEL
LIN {X 0,Y 326.623,Z 246.302,A -85,B 0,C 180,E1 -14964.125,E2 -14964.125} C_VEL
LIN {X 0,Y 326.656,Z 246.295,A -85,B 0,C 180,E1 -14966.854,E2 -14966.854} C_VEL
LIN {X 0,Y 326.605,Z 246.304,A -85,B 0,C 180,E1 -14970.606,E2 -14970.606} C_VEL
LIN {X 0,Y 326.576,Z 246.306,A -85,B 0,C 180,E1 -14974.016,E2 -14974.016} C_VEL
LIN {X 0,Y 326.606,Z 246.297,A -85,B 0,C 180,E1 -14977.86,E2 -14977.86} C_VEL
LIN {X 0,Y 326.663,Z 246.627,A -85,B 0,C 180,E1 -14978.502,E2 -14978.502} C_VEL
LIN {X 0,Y 328.99,Z 255.789,A -85,B 0,C 180,E1 -14981.614,E2 -14981.614} C_VEL
LIN {X 0,Y 329.889,Z 259.869,A -85,B 0,C 180,E1 -14982.866,E2 -14982.866} C_VEL
LIN {X 0,Y 336.246,Z 274.276,A -85,B 0,C 180,E1 -14983.912,E2 -14983.912} C_VEL
LIN {X 0,Y 337.6,Z 278.905,A -85,B 0,C 180,E1 -14984.157,E2 -14984.157} C_VEL
LIN {X 0,Y 340.563,Z 293.204,A -85,B 0,C 180,E1 -14984.784,E2 -14984.784} C_VEL
LIN {X 0,Y 338.456,Z 368.247,A -85,B 0,C 180,E1 -14986.452,E2 -14986.452} C_VEL
LIN {X 0,Y 337.614,Z 381.689,A -85,B 0,C 180,E1 -14986.997,E2 -14986.997} C_VEL
LIN {X 0,Y 336.507,Z 394.354,A -85,B 0,C 180,E1 -14987.763,E2 -14987.763} C_VEL
LIN {X 0,Y 335.091,Z 406.643,A -85,B 0,C 180,E1 -14988.78,E2 -14988.78} C_VEL
LIN {X 0,Y 333.518,Z 418.115,A -85,B 0,C 180,E1 -14990.009,E2 -14990.009} C_VEL
LIN {X 0,Y 332.09,Z 427.12,A -85,B 0,C 180,E1 -14991.211,E2 -14991.211} C_VEL
LIN {X 0,Y 330.582,Z 436.26,A -85,B 0,C 180,E1 -14992.71,E2 -14992.71} C_VEL
LIN {X 0,Y 329.091,Z 444.915,A -85,B 0,C 180,E1 -14994.475,E2 -14994.475} C_VEL
LIN {X 0,Y 327.683,Z 452.949,A -85,B 0,C 180,E1 -14996.528,E2 -14996.528} C_VEL
LIN {X 0,Y 326.766,Z 458.134,A -85,B 0,C 180,E1 -14998.204,E2 -14998.204} C_VEL
LIN {X 0,Y 325.961,Z 463.168,A -85,B 0,C 180,E1 -15000.273,E2 -15000.273} C_VEL
LIN {X 0,Y 325.377,Z 466.807,A -85,B 0,C 180,E1 -15002.309,E2 -15002.309} C_VEL
LIN {X 0,Y 324.898,Z 469.309,A -85,B 0,C 180,E1 -15004.368,E2 -15004.368} C_VEL
LIN {X 0,Y 324.698,Z 470.34,A -85,B 0,C 180,E1 -15005.719,E2 -15005.719} C_VEL
LIN {X 0,Y 324.561,Z 470.916,A -85,B 0,C 180,E1 -15007.062,E2 -15007.062} C_VEL
LIN {X 0,Y 324.554,Z 470.959,A -85,B 0,C 180,E1 -15008.594,E2 -15008.594} C_VEL
LIN {X 0,Y 324.579,Z 469.831,A -85,B 0,C 180,E1 -15011.049,E2 -15011.049} C_VEL
LIN {X 0,Y 324.66,Z 468.544,A -85,B 0,C 180,E1 -15012.361,E2 -15012.361} C_VEL
LIN {X 0,Y 324.94,Z 465.78,A -85,B 0,C 180,E1 -15014.317,E2 -15014.317} C_VEL
LIN {X 0,Y 325.327,Z 461.567,A -85,B 0,C 180,E1 -15016.411,E2 -15016.411} C_VEL
LIN {X 0,Y 325.763,Z 456.904,A -85,B 0,C 180,E1 -15018.175,E2 -15018.175} C_VEL
LIN {X 0,Y 326.362,Z 450.564,A -85,B 0,C 180,E1 -15020.082,E2 -15020.082} C_VEL
LIN {X 0,Y 327.29,Z 442.528,A -85,B 0,C 180,E1 -15021.996,E2 -15021.996} C_VEL
LIN {X 0,Y 328.242,Z 434.444,A -85,B 0,C 180,E1 -15023.548,E2 -15023.548} C_VEL
LIN {X 0,Y 329.305,Z 424.491,A -85,B 0,C 180,E1 -15025.105,E2 -15025.105} C_VEL
LIN {X 0,Y 330.438,Z 414.652,A -85,B 0,C 180,E1 -15026.344,E2 -15026.344} C_VEL
LIN {X 0,Y 331.464,Z 403.43,A -85,B 0,C 180,E1 -15027.478,E2 -15027.478} C_VEL
LIN {X 0,Y 332.365,Z 391.407,A -85,B 0,C 180,E1 -15028.412,E2 -15028.412} C_VEL
LIN {X 0,Y 333.182,Z 378.677,A -85,B 0,C 180,E1 -15029.133,E2 -15029.133} C_VEL
LIN {X 0,Y 333.683,Z 365.478,A -85,B 0,C 180,E1 -15029.625,E2 -15029.625} C_VEL
LIN {X 0,Y 335.106,Z 290.182,A -85,B 0,C 180,E1 -15031.27,E2 -15031.27} C_VEL
LIN {X 0,Y 330.409,Z 263.21,A -85,B 0,C 180,E1 -15032.165,E2 -15032.165} C_VEL
LIN {X 0,Y 329.35,Z 259.762,A -85,B 0,C 180,E1 -15032.381,E2 -15032.381} C_VEL
LIN {X 0,Y 328.059,Z 253.205,A -85,B 0,C 180,E1 -15034.302,E2 -15034.302} C_VEL
LIN {X 0,Y 326.94,Z 246.315,A -85,B 0,C 180,E1 -15036.482,E2 -15036.482} C_VEL
LIN {X 0,Y 326.769,Z 246.281,A -85,B 0,C 180,E1 -15039.909,E2 -15039.909} C_VEL
LIN {X 0,Y 326.721,Z 246.29,A -85,B 0,C 180,E1 -15043.689,E2 -15043.689} C_VEL
LIN {X 0,Y 326.663,Z 246.29,A -85,B 0,C 180,E1 -15047.532,E2 -15047.532} C_VEL
LIN {X 0,Y 326.62,Z 246.3,A -85,B 0,C 180,E1 -15050.14,E2 -15050.14} C_VEL
LIN {X 0,Y 326.582,Z 246.306,A -85,B 0,C 180,E1 -15054.136,E2 -15054.136} C_VEL
LIN {X 0,Y 326.568,Z 246.309,A -85,B 0,C 180,E1 -15058.261,E2 -15058.261} C_VEL
LIN {X 0,Y 326.541,Z 246.306,A -85,B 0,C 180,E1 -15061.102,E2 -15061.102} C_VEL
LIN {X 0,Y 326.569,Z 246.302,A -85,B 0,C 180,E1 -15064.32,E2 -15064.32} C_VEL
LIN {X 0,Y 325.909,Z 246.386,A -85,B 0,C 180,E1 -15065.349,E2 -15065.349} C_VEL
LIN {X 0,Y 323.091,Z 246.736,A -85,B 0,C 180,E1 -15067.026,E2 -15067.026} C_VEL
LIN {X 0,Y 320.676,Z 247.041,A -85,B 0,C 180,E1 -15068.384,E2 -15068.384} C_VEL
LIN {X 0,Y 319.602,Z 247.168,A -85,B 0,C 180,E1 -15069.434,E2 -15069.434} C_VEL
LIN {X 0,Y 319.494,Z 247.179,A -85,B 0,C 180,E1 -15069.79,E2 -15069.79} C_VEL
LIN {X 0,Y 319.497,Z 247.184,A -85,B 0,C 180,E1 -15073.465,E2 -15073.465} C_VEL
LIN {X 0,Y 319.532,Z 247.179,A -85,B 0,C 180,E1 -15077.022,E2 -15077.022} C_VEL
LIN {X 0,Y 319.529,Z 247.176,A -85,B 0,C 180,E1 -15080.376,E2 -15080.376} C_VEL
LIN {X 0,Y 319.564,Z 247.177,A -85,B 0,C 180,E1 -15084.464,E2 -15084.464} C_VEL
LIN {X 0,Y 319.511,Z 247.178,A -85,B 0,C 180,E1 -15088.143,E2 -15088.143} C_VEL
LIN {X 0,Y 319.534,Z 247.177,A -85,B 0,C 180,E1 -15091.619,E2 -15091.619} C_VEL
LIN {X 0,Y 319.534,Z 247.184,A -85,B 0,C 180,E1 -15095.305,E2 -15095.305} C_VEL
LIN {X 0,Y 319.559,Z 247.176,A -85,B 0,C 180,E1 -15098.051,E2 -15098.051} C_VEL
LIN {X 0,Y 319.611,Z 247.163,A -85,B 0,C 180,E1 -15102.076,E2 -15102.076} C_VEL
LIN {X 0,Y 319.732,Z 247.155,A -85,B 0,C 180,E1 -15106.013,E2 -15106.013} C_VEL
LIN {X 0,Y 319.736,Z 247.159,A -85,B 0,C 180,E1 -15109.878,E2 -15109.878} C_VEL
LIN {X 0,Y 319.901,Z 247.135,A -85,B 0,C 180,E1 -15113.699,E2 -15113.699} C_VEL
LIN {X 0,Y 319.961,Z 247.119,A -85,B 0,C 180,E1 -15117.487,E2 -15117.487} C_VEL
LIN {X 0,Y 320.018,Z 247.118,A -85,B 0,C 180,E1 -15121.263,E2 -15121.263} C_VEL
LIN {X 0,Y 319.907,Z 247.136,A -85,B 0,C 180,E1 -15126.311,E2 -15126.311} C_VEL
LIN {X 0,Y 319.746,Z 247.147,A -85,B 0,C 180,E1 -15130.132,E2 -15130.132} C_VEL
LIN {X 0,Y 319.746,Z 247.153,A -85,B 0,C 180,E1 -15133.996,E2 -15133.996} C_VEL
LIN {X 0,Y 319.629,Z 247.166,A -85,B 0,C 180,E1 -15137.933,E2 -15137.933} C_VEL
LIN {X 0,Y 319.581,Z 247.17,A -85,B 0,C 180,E1 -15141.958,E2 -15141.958} C_VEL
LIN {X 0,Y 319.583,Z 247.173,A -85,B 0,C 180,E1 -15146.097,E2 -15146.097} C_VEL
LIN {X 0,Y 319.558,Z 247.178,A -85,B 0,C 180,E1 -15148.941,E2 -15148.941} C_VEL
LIN {X 0,Y 319.541,Z 247.178,A -85,B 0,C 180,E1 -15151.865,E2 -15151.865} C_VEL
LIN {X 0,Y 319.597,Z 247.172,A -85,B 0,C 180,E1 -15155.545,E2 -15155.545} C_VEL
LIN {X 0,Y 319.546,Z 247.182,A -85,B 0,C 180,E1 -15159.664,E2 -15159.664} C_VEL
LIN {X 0,Y 319.535,Z 247.181,A -85,B 0,C 180,E1 -15163.461,E2 -15163.461} C_VEL
LIN {X 0,Y 319.567,Z 247.174,A -85,B 0,C 180,E1 -15167.017,E2 -15167.017} C_VEL
LIN {X 0,Y 319.533,Z 247.179,A -85,B 0,C 180,E1 -15170.367,E2 -15170.367} C_VEL
LIN {X 0,Y 319.597,Z 247.172,A -85,B 0,C 180,E1 -15174.458,E2 -15174.458} C_VEL
LIN {X 0,Y 319.542,Z 247.181,A -85,B 0,C 180,E1 -15178.137,E2 -15178.137} C_VEL
LIN {X 0,Y 319.633,Z 247.302,A -85,B 0,C 180,E1 -15180.165,E2 -15180.165} C_VEL
LIN {X 0,Y 322.018,Z 258.936,A -85,B 0,C 180,E1 -15183.724,E2 -15183.724} C_VEL
LIN {X 0,Y 323.027,Z 265.353,A -85,B 0,C 180,E1 -15185.581,E2 -15185.581} C_VEL
LIN {X 0,Y 322.847,Z 268.159,A -85,B 0,C 180,E1 -15186.274,E2 -15186.274} C_VEL
LIN {X 0,Y 323.883,Z 274.918,A -85,B 0,C 180,E1 -15186.552,E2 -15186.552} C_VEL
LIN {X 0,Y 328.343,Z 304.854,A -85,B 0,C 180,E1 -15187.511,E2 -15187.511} C_VEL
LIN {X 0,Y 326.857,Z 375.657,A -85,B 0,C 180,E1 -15189.095,E2 -15189.095} C_VEL
LIN {X 0,Y 326.18,Z 388.959,A -85,B 0,C 180,E1 -15189.626,E2 -15189.626} C_VEL
LIN {X 0,Y 325.253,Z 402.311,A -85,B 0,C 180,E1 -15190.43,E2 -15190.43} C_VEL
LIN {X 0,Y 324.217,Z 413.512,A -85,B 0,C 180,E1 -15191.351,E2 -15191.351} C_VEL
LIN {X 0,Y 322.966,Z 425.159,A -85,B 0,C 180,E1 -15192.588,E2 -15192.588} C_VEL
LIN {X 0,Y 321.882,Z 436.093,A -85,B 0,C 180,E1 -15194.063,E2 -15194.063} C_VEL
LIN {X 0,Y 320.691,Z 445.889,A -85,B 0,C 180,E1 -15195.725,E2 -15195.725} C_VEL
LIN {X 0,Y 319.6,Z 454.839,A -85,B 0,C 180,E1 -15197.618,E2 -15197.618} C_VEL
LIN {X 0,Y 318.855,Z 462.011,A -85,B 0,C 180,E1 -15199.521,E2 -15199.521} C_VEL
LIN {X 0,Y 318.23,Z 468.527,A -85,B 0,C 180,E1 -15201.745,E2 -15201.745} C_VEL
LIN {X 0,Y 317.928,Z 472.814,A -85,B 0,C 180,E1 -15203.652,E2 -15203.652} C_VEL
LIN {X 0,Y 317.818,Z 475.081,A -85,B 0,C 180,E1 -15204.923,E2 -15204.923} C_VEL
LIN {X 0,Y 317.782,Z 476.878,A -85,B 0,C 180,E1 -15206.194,E2 -15206.194} C_VEL
LIN {X 0,Y 317.736,Z 478.229,A -85,B 0,C 180,E1 -15207.463,E2 -15207.463} C_VEL
LIN {X 0,Y 317.699,Z 479.181,A -85,B 0,C 180,E1 -15208.73,E2 -15208.73} C_VEL
LIN {X 0,Y 317.712,Z 479.744,A -85,B 0,C 180,E1 -15209.998,E2 -15209.998} C_VEL
LIN {X 0,Y 317.698,Z 479.88,A -85,B 0,C 180,E1 -15211.266,E2 -15211.266} C_VEL
LIN {X 0,Y 317.737,Z 479.61,A -85,B 0,C 180,E1 -15212.533,E2 -15212.533} C_VEL
LIN {X 0,Y 317.795,Z 478.957,A -85,B 0,C 180,E1 -15213.802,E2 -15213.802} C_VEL
LIN {X 0,Y 317.909,Z 477.098,A -85,B 0,C 180,E1 -15215.812,E2 -15215.812} C_VEL
LIN {X 0,Y 318.383,Z 473.459,A -85,B 0,C 180,E1 -15218.247,E2 -15218.247} C_VEL
LIN {X 0,Y 318.988,Z 469.435,A -85,B 0,C 180,E1 -15220.15,E2 -15220.15} C_VEL
LIN {X 0,Y 320.047,Z 463.276,A -85,B 0,C 180,E1 -15222.361,E2 -15222.361} C_VEL
LIN {X 0,Y 321.333,Z 456.587,A -85,B 0,C 180,E1 -15224.242,E2 -15224.242} C_VEL
LIN {X 0,Y 322.938,Z 448.31,A -85,B 0,C 180,E1 -15226.107,E2 -15226.107} C_VEL
LIN {X 0,Y 324.338,Z 439.831,A -85,B 0,C 180,E1 -15227.657,E2 -15227.657} C_VEL
LIN {X 0,Y 326.079,Z 429.392,A -85,B 0,C 180,E1 -15229.187,E2 -15229.187} C_VEL
LIN {X 0,Y 327.71,Z 419.077,A -85,B 0,C 180,E1 -15230.393,E2 -15230.393} C_VEL
LIN {X 0,Y 329.27,Z 407.787,A -85,B 0,C 180,E1 -15231.437,E2 -15231.437} C_VEL
LIN {X 0,Y 330.451,Z 396.248,A -85,B 0,C 180,E1 -15232.259,E2 -15232.259} C_VEL
LIN {X 0,Y 331.606,Z 383.044,A -85,B 0,C 180,E1 -15232.917,E2 -15232.917} C_VEL
LIN {X 0,Y 332.29,Z 370.286,A -85,B 0,C 180,E1 -15233.32,E2 -15233.32} C_VEL
LIN {X 0,Y 333.932,Z 305.681,A -85,B 0,C 180,E1 -15234.769,E2 -15234.769} C_VEL
LIN {X 0,Y 330.409,Z 286.723,A -85,B 0,C 180,E1 -15235.589,E2 -15235.589} C_VEL
LIN {X 0,Y 327.65,Z 275.46,A -85,B 0,C 180,E1 -15236.158,E2 -15236.158} C_VEL
LIN {X 0,Y 324.315,Z 267.61,A -85,B 0,C 180,E1 -15236.762,E2 -15236.762} C_VEL
LIN {X 0,Y 322.402,Z 258.601,A -85,B 0,C 180,E1 -15239.606,E2 -15239.606} C_VEL
LIN {X 0,Y 319.992,Z 249.018,A -85,B 0,C 180,E1 -15242.925,E2 -15242.925} C_VEL
LIN {X 0,Y 319.572,Z 247.205,A -85,B 0,C 180,E1 -15243.681,E2 -15243.681} C_VEL
LIN {X 0,Y 319.561,Z 247.179,A -85,B 0,C 180,E1 -15246.424,E2 -15246.424} C_VEL
LIN {X 0,Y 319.564,Z 247.178,A -85,B 0,C 180,E1 -15249.665,E2 -15249.665} C_VEL
LIN {X 0,Y 319.524,Z 247.18,A -85,B 0,C 180,E1 -15253.456,E2 -15253.456} C_VEL
LIN {X 0,Y 319.554,Z 247.161,A -85,B 0,C 180,E1 -15257.012,E2 -15257.012} C_VEL
LIN {X 0,Y 319.516,Z 247.182,A -85,B 0,C 180,E1 -15260.362,E2 -15260.362} C_VEL
LIN {X 0,Y 319.579,Z 247.173,A -85,B 0,C 180,E1 -15264.453,E2 -15264.453} C_VEL
LIN {X 0,Y 319.523,Z 247.18,A -85,B 0,C 180,E1 -15268.133,E2 -15268.133} C_VEL
LIN {X 0,Y 319.569,Z 247.175,A -85,B 0,C 180,E1 -15271.599,E2 -15271.599} C_VEL
LIN {X 0,Y 319.538,Z 247.176,A -85,B 0,C 180,E1 -15275.294,E2 -15275.294} C_VEL
LIN {X 0,Y 319.56,Z 247.175,A -85,B 0,C 180,E1 -15278.041,E2 -15278.041} C_VEL
LIN {X 0,Y 319.608,Z 247.17,A -85,B 0,C 180,E1 -15282.066,E2 -15282.066} C_VEL
LIN {X 0,Y 319.724,Z 247.157,A -85,B 0,C 180,E1 -15286.003,E2 -15286.003} C_VEL
LIN {X 0,Y 319.725,Z 247.158,A -85,B 0,C 180,E1 -15289.867,E2 -15289.867} C_VEL
LIN {X 0,Y 319.896,Z 247.134,A -85,B 0,C 180,E1 -15293.689,E2 -15293.689} C_VEL
LIN {X 0,Y 319.998,Z 247.123,A -85,B 0,C 180,E1 -15298.737,E2 -15298.737} C_VEL
LIN {X 0,Y 319.941,Z 247.129,A -85,B 0,C 180,E1 -15302.513,E2 -15302.513} C_VEL
LIN {X 0,Y 319.869,Z 247.136,A -85,B 0,C 180,E1 -15306.427,E2 -15306.427} C_VEL
LIN {X 0,Y 319.717,Z 247.154,A -85,B 0,C 180,E1 -15310.123,E2 -15310.123} C_VEL
LIN {X 0,Y 319.712,Z 247.156,A -85,B 0,C 180,E1 -15313.988,E2 -15313.988} C_VEL
LIN {X 0,Y 319.602,Z 247.174,A -85,B 0,C 180,E1 -15317.924,E2 -15317.924} C_VEL
LIN {X 0,Y 319.543,Z 247.18,A -85,B 0,C 180,E1 -15321.95,E2 -15321.95} C_VEL
LIN {X 0,Y 319.607,Z 247.173,A -85,B 0,C 180,E1 -15326.084,E2 -15326.084} C_VEL
LIN {X 0,Y 319.551,Z 247.165,A -85,B 0,C 180,E1 -15328.931,E2 -15328.931} C_VEL
LIN {X 0,Y 319.501,Z 247.179,A -85,B 0,C 180,E1 -15331.858,E2 -15331.858} C_VEL
LIN {X 0,Y 319.549,Z 247.172,A -85,B 0,C 180,E1 -15335.539,E2 -15335.539} C_VEL
LIN {X 0,Y 319.598,Z 247.381,A -85,B 0,C 180,E1 -15337.77,E2 -15337.77} C_VEL
LIN {X 0,Y 322.237,Z 257.809,A -85,B 0,C 180,E1 -15341.441,E2 -15341.441} C_VEL
LIN {X 0,Y 322.809,Z 260.189,A -85,B 0,C 180,E1 -15342.125,E2 -15342.125} C_VEL
LIN {X 0,Y 329.902,Z 275.903,A -85,B 0,C 180,E1 -15343.323,E2 -15343.323} C_VEL
LIN {X 0,Y 331.4,Z 280.126,A -85,B 0,C 180,E1 -15343.582,E2 -15343.582} C_VEL
LIN {X 0,Y 334.258,Z 293.817,A -85,B 0,C 180,E1 -15344.204,E2 -15344.204} C_VEL
LIN {X 0,Y 332.149,Z 368.194,A -85,B 0,C 180,E1 -15345.892,E2 -15345.892} C_VEL
LIN {X 0,Y 331.271,Z 381.783,A -85,B 0,C 180,E1 -15346.451,E2 -15346.451} C_VEL
LIN {X 0,Y 330.175,Z 393.708,A -85,B 0,C 180,E1 -15347.174,E2 -15347.174} C_VEL
LIN {X 0,Y 328.884,Z 405.087,A -85,B 0,C 180,E1 -15348.107,E2 -15348.107} C_VEL
LIN {X 0,Y 327.28,Z 416.331,A -85,B 0,C 180,E1 -15349.29,E2 -15349.29} C_VEL
LIN {X 0,Y 325.602,Z 426.77,A -85,B 0,C 180,E1 -15350.674,E2 -15350.674} C_VEL
LIN {X 0,Y 323.966,Z 436.067,A -85,B 0,C 180,E1 -15352.207,E2 -15352.207} C_VEL
LIN {X 0,Y 322.391,Z 444.525,A -85,B 0,C 180,E1 -15353.946,E2 -15353.946} C_VEL
LIN {X 0,Y 320.971,Z 452.214,A -85,B 0,C 180,E1 -15355.922,E2 -15355.922} C_VEL
LIN {X 0,Y 320.068,Z 457.05,A -85,B 0,C 180,E1 -15357.457,E2 -15357.457} C_VEL
LIN {X 0,Y 319.119,Z 462.359,A -85,B 0,C 180,E1 -15359.57,E2 -15359.57} C_VEL
LIN {X 0,Y 318.669,Z 465.144,A -85,B 0,C 180,E1 -15360.977,E2 -15360.977} C_VEL
LIN {X 0,Y 318.26,Z 467.327,A -85,B 0,C 180,E1 -15362.374,E2 -15362.374} C_VEL
LIN {X 0,Y 317.917,Z 469.024,A -85,B 0,C 180,E1 -15363.763,E2 -15363.763} C_VEL
LIN {X 0,Y 317.705,Z 470.183,A -85,B 0,C 180,E1 -15365.149,E2 -15365.149} C_VEL
LIN {X 0,Y 317.497,Z 470.875,A -85,B 0,C 180,E1 -15366.522,E2 -15366.522} C_VEL
LIN {X 0,Y 317.45,Z 471.073,A -85,B 0,C 180,E1 -15368.39,E2 -15368.39} C_VEL
LIN {X 0,Y 317.445,Z 470.198,A -85,B 0,C 180,E1 -15370.607,E2 -15370.607} C_VEL
LIN {X 0,Y 317.552,Z 468.941,A -85,B 0,C 180,E1 -15372.091,E2 -15372.091} C_VEL
LIN {X 0,Y 317.793,Z 466.534,A -85,B 0,C 180,E1 -15373.954,E2 -15373.954} C_VEL
LIN {X 0,Y 318.235,Z 462.074,A -85,B 0,C 180,E1 -15376.309,E2 -15376.309} C_VEL
LIN {X 0,Y 318.765,Z 456.243,A -85,B 0,C 180,E1 -15378.557,E2 -15378.557} C_VEL
LIN {X 0,Y 319.462,Z 449.694,A -85,B 0,C 180,E1 -15380.505,E2 -15380.505} C_VEL
LIN {X 0,Y 320.418,Z 441.47,A -85,B 0,C 180,E1 -15382.44,E2 -15382.44} C_VEL
LIN {X 0,Y 321.406,Z 433.07,A -85,B 0,C 180,E1 -15384.04,E2 -15384.04} C_VEL
LIN {X 0,Y 322.621,Z 422.763,A -85,B 0,C 180,E1 -15385.629,E2 -15385.629} C_VEL
LIN {X 0,Y 323.732,Z 412.719,A -85,B 0,C 180,E1 -15386.865,E2 -15386.865} C_VEL
LIN {X 0,Y 324.804,Z 401.293,A -85,B 0,C 180,E1 -15387.987,E2 -15387.987} C_VEL
LIN {X 0,Y 325.693,Z 390.027,A -85,B 0,C 180,E1 -15388.843,E2 -15388.843} C_VEL
LIN {X 0,Y 326.438,Z 377.584,A -85,B 0,C 180,E1 -15389.539,E2 -15389.539} C_VEL
LIN {X 0,Y 326.937,Z 364.785,A -85,B 0,C 180,E1 -15390.002,E2 -15390.002} C_VEL
LIN {X 0,Y 328.4,Z 291.153,A -85,B 0,C 180,E1 -15391.638,E2 -15391.638} C_VEL
LIN {X 0,Y 324.005,Z 265.526,A -85,B 0,C 180,E1 -15392.508,E2 -15392.508} C_VEL
LIN {X 0,Y 322.308,Z 260.059,A -85,B 0,C 180,E1 -15392.783,E2 -15392.783} C_VEL
LIN {X 0,Y 319.925,Z 247.474,A -85,B 0,C 180,E1 -15396.625,E2 -15396.625} C_VEL
LIN {X 0,Y 319.874,Z 247.14,A -85,B 0,C 180,E1 -15396.943,E2 -15396.943} C_VEL
LIN {X 0,Y 319.716,Z 247.159,A -85,B 0,C 180,E1 -15400.13,E2 -15400.13} C_VEL
LIN {X 0,Y 319.695,Z 247.158,A -85,B 0,C 180,E1 -15404.727,E2 -15404.727} C_VEL
LIN {X 0,Y 319.655,Z 247.164,A -85,B 0,C 180,E1 -15409.041,E2 -15409.041} C_VEL
LIN {X 0,Y 319.511,Z 247.183,A -85,B 0,C 180,E1 -15413.326,E2 -15413.326} C_VEL
LIN {X 0,Y 319.523,Z 247.184,A -85,B 0,C 180,E1 -15416.1,E2 -15416.1} C_VEL
LIN {X 0,Y 319.512,Z 247.183,A -85,B 0,C 180,E1 -15418.943,E2 -15418.943} C_VEL
LIN {X 0,Y 319.493,Z 247.186,A -85,B 0,C 180,E1 -15421.868,E2 -15421.868} C_VEL
LIN {X 0,Y 319.551,Z 247.177,A -85,B 0,C 180,E1 -15425.547,E2 -15425.547} C_VEL
LIN {X 0,Y 319.505,Z 247.179,A -85,B 0,C 180,E1 -15429.667,E2 -15429.667} C_VEL
LIN {X 0,Y 319.494,Z 247.179,A -85,B 0,C 180,E1 -15429.79,E2 -15429.79} C_VEL
LIN {X 0,Y 318.763,Z 247.277,A -85,B 0,C 180,E1 -15430.841,E2 -15430.841} C_VEL
LIN {X 0,Y 315.873,Z 247.639,A -85,B 0,C 180,E1 -15432.552,E2 -15432.552} C_VEL
LIN {X 0,Y 313.476,Z 247.934,A -85,B 0,C 180,E1 -15433.939,E2 -15433.939} C_VEL
LIN {X 0,Y 312.475,Z 248.061,A -85,B 0,C 180,E1 -15435.012,E2 -15435.012} C_VEL
LIN {X 0,Y 312.407,Z 248.064,A -85,B 0,C 180,E1 -15435.376,E2 -15435.376} C_VEL
LIN {X 0,Y 312.436,Z 248.059,A -85,B 0,C 180,E1 -15437.931,E2 -15437.931} C_VEL
LIN {X 0,Y 312.467,Z 248.058,A -85,B 0,C 180,E1 -15441.929,E2 -15441.929} C_VEL
LIN {X 0,Y 312.515,Z 248.054,A -85,B 0,C 180,E1 -15444.226,E2 -15444.226} C_VEL
LIN {X 0,Y 312.489,Z 248.056,A -85,B 0,C 180,E1 -15447.339,E2 -15447.339} C_VEL
LIN {X 0,Y 312.474,Z 248.056,A -85,B 0,C 180,E1 -15451.306,E2 -15451.306} C_VEL
LIN {X 0,Y 312.514,Z 248.053,A -85,B 0,C 180,E1 -15454.711,E2 -15454.711} C_VEL
LIN {X 0,Y 312.535,Z 248.055,A -85,B 0,C 180,E1 -15457.531,E2 -15457.531} C_VEL
LIN {X 0,Y 312.564,Z 248.043,A -85,B 0,C 180,E1 -15461.658,E2 -15461.658} C_VEL
LIN {X 0,Y 312.685,Z 248.031,A -85,B 0,C 180,E1 -15465.692,E2 -15465.692} C_VEL
LIN {X 0,Y 312.686,Z 248.036,A -85,B 0,C 180,E1 -15469.647,E2 -15469.647} C_VEL
LIN {X 0,Y 312.799,Z 248.018,A -85,B 0,C 180,E1 -15472.258,E2 -15472.258} C_VEL
LIN {X 0,Y 312.691,Z 248.025,A -85,B 0,C 180,E1 -15474.847,E2 -15474.847} C_VEL
LIN {X 0,Y 312.973,Z 247.993,A -85,B 0,C 180,E1 -15478.718,E2 -15478.718} C_VEL
LIN {X 0,Y 312.985,Z 247.994,A -85,B 0,C 180,E1 -15481.292,E2 -15481.292} C_VEL
LIN {X 0,Y 312.849,Z 248.013,A -85,B 0,C 180,E1 -15486.454,E2 -15486.454} C_VEL
LIN {X 0,Y 312.697,Z 248.026,A -85,B 0,C 180,E1 -15490.363,E2 -15490.363} C_VEL
LIN {X 0,Y 312.682,Z 248.036,A -85,B 0,C 180,E1 -15494.869,E2 -15494.869} C_VEL
LIN {X 0,Y 312.563,Z 248.044,A -85,B 0,C 180,E1 -15499.196,E2 -15499.196} C_VEL
LIN {X 0,Y 312.538,Z 248.052,A -85,B 0,C 180,E1 -15502.781,E2 -15502.781} C_VEL
LIN {X 0,Y 312.544,Z 248.05,A -85,B 0,C 180,E1 -15505.91,E2 -15505.91} C_VEL
LIN {X 0,Y 312.512,Z 248.051,A -85,B 0,C 180,E1 -15509.658,E2 -15509.658} C_VEL
LIN {X 0,Y 312.538,Z 248.052,A -85,B 0,C 180,E1 -15513.691,E2 -15513.691} C_VEL
LIN {X 0,Y 312.528,Z 248.053,A -85,B 0,C 180,E1 -15517.389,E2 -15517.389} C_VEL
LIN {X 0,Y 312.458,Z 248.061,A -85,B 0,C 180,E1 -15520.719,E2 -15520.719} C_VEL
LIN {X 0,Y 312.467,Z 248.061,A -85,B 0,C 180,E1 -15524.212,E2 -15524.212} C_VEL
LIN {X 0,Y 312.472,Z 248.063,A -85,B 0,C 180,E1 -15527.926,E2 -15527.926} C_VEL
LIN {X 0,Y 312.494,Z 248.057,A -85,B 0,C 180,E1 -15531.925,E2 -15531.925} C_VEL
LIN {X 0,Y 312.549,Z 248.052,A -85,B 0,C 180,E1 -15534.22,E2 -15534.22} C_VEL
LIN {X 0,Y 312.52,Z 248.056,A -85,B 0,C 180,E1 -15537.334,E2 -15537.334} C_VEL
LIN {X 0,Y 312.588,Z 248.255,A -85,B 0,C 180,E1 -15539.888,E2 -15539.888} C_VEL
LIN {X 0,Y 314.966,Z 259.829,A -85,B 0,C 180,E1 -15543.493,E2 -15543.493} C_VEL
LIN {X 0,Y 316.06,Z 266.546,A -85,B 0,C 180,E1 -15545.486,E2 -15545.486} C_VEL
LIN {X 0,Y 316.022,Z 268.373,A -85,B 0,C 180,E1 -15545.861,E2 -15545.861} C_VEL
LIN {X 0,Y 320.56,Z 298.099,A -85,B 0,C 180,E1 -15546.899,E2 -15546.899} C_VEL
LIN {X 0,Y 321.589,Z 306.152,A -85,B 0,C 180,E1 -15547.151,E2 -15547.151} C_VEL
LIN {X 0,Y 320.04,Z 376.266,A -85,B 0,C 180,E1 -15548.754,E2 -15548.754} C_VEL
LIN {X 0,Y 319.346,Z 389.338,A -85,B 0,C 180,E1 -15549.297,E2 -15549.297} C_VEL
LIN {X 0,Y 318.434,Z 402.014,A -85,B 0,C 180,E1 -15550.078,E2 -15550.078} C_VEL
LIN {X 0,Y 317.285,Z 414.076,A -85,B 0,C 180,E1 -15551.096,E2 -15551.096} C_VEL
LIN {X 0,Y 316.003,Z 425.61,A -85,B 0,C 180,E1 -15552.359,E2 -15552.359} C_VEL
LIN {X 0,Y 314.896,Z 436.389,A -85,B 0,C 180,E1 -15553.858,E2 -15553.858} C_VEL
LIN {X 0,Y 313.753,Z 445.329,A -85,B 0,C 180,E1 -15555.402,E2 -15555.402} C_VEL
LIN {X 0,Y 312.646,Z 454.366,A -85,B 0,C 180,E1 -15557.338,E2 -15557.338} C_VEL
LIN {X 0,Y 311.833,Z 461.625,A -85,B 0,C 180,E1 -15559.282,E2 -15559.282} C_VEL
LIN {X 0,Y 311.33,Z 466.508,A -85,B 0,C 180,E1 -15560.906,E2 -15560.906} C_VEL
LIN {X 0,Y 310.942,Z 471.24,A -85,B 0,C 180,E1 -15562.857,E2 -15562.857} C_VEL
LIN {X 0,Y 310.726,Z 474.838,A -85,B 0,C 180,E1 -15564.807,E2 -15564.807} C_VEL
LIN {X 0,Y 310.697,Z 476.681,A -85,B 0,C 180,E1 -15566.107,E2 -15566.107} C_VEL
LIN {X 0,Y 310.661,Z 478.055,A -85,B 0,C 180,E1 -15567.405,E2 -15567.405} C_VEL
LIN {X 0,Y 310.616,Z 479.029,A -85,B 0,C 180,E1 -15568.702,E2 -15568.702} C_VEL
LIN {X 0,Y 310.626,Z 479.613,A -85,B 0,C 180,E1 -15569.998,E2 -15569.998} C_VEL
LIN {X 0,Y 310.615,Z 479.791,A -85,B 0,C 180,E1 -15571.294,E2 -15571.294} C_VEL
LIN {X 0,Y 310.662,Z 479.544,A -85,B 0,C 180,E1 -15572.591,E2 -15572.591} C_VEL
LIN {X 0,Y 310.711,Z 478.914,A -85,B 0,C 180,E1 -15573.889,E2 -15573.889} C_VEL
LIN {X 0,Y 310.822,Z 477.3,A -85,B 0,C 180,E1 -15575.771,E2 -15575.771} C_VEL
LIN {X 0,Y 311.332,Z 473.536,A -85,B 0,C 180,E1 -15578.435,E2 -15578.435} C_VEL
LIN {X 0,Y 311.988,Z 469.567,A -85,B 0,C 180,E1 -15580.38,E2 -15580.38} C_VEL
LIN {X 0,Y 312.971,Z 464.479,A -85,B 0,C 180,E1 -15582.315,E2 -15582.315} C_VEL
LIN {X 0,Y 314.2,Z 458.095,A -85,B 0,C 180,E1 -15584.242,E2 -15584.242} C_VEL
LIN {X 0,Y 315.852,Z 450.148,A -85,B 0,C 180,E1 -15586.147,E2 -15586.147} C_VEL
LIN {X 0,Y 317.25,Z 442.214,A -85,B 0,C 180,E1 -15587.707,E2 -15587.707} C_VEL
LIN {X 0,Y 318.855,Z 433.325,A -85,B 0,C 180,E1 -15589.137,E2 -15589.137} C_VEL
